# B&R Automation Studio project BaseProject (part 5)

#### Main.st - Init, cyclic, exit code
```iecst
// --------------------------------------------------------------------------------------------------------------------
// Logbook Task
// This task reads the PLC logbook and creates the data structure to display it in mappView
// --------------------------------------------------------------------------------------------------------------------
PROGRAM _INIT
	// Set time range to all on startup
	DTGetTime_0.enable := TRUE;
	DTGetTime_0();
	LogbookInterface.Par.FilterDateStart := STRING_TO_DATE('D#1999-12-31');
	LogbookInterface.Par.FilterDateEnd := DT_TO_DATE(DTGetTime_0.DT1);

	// Read data after reboot
	LogbookInterface.Cmd.Refresh := TRUE;

	// define what object type should be searched for
	LogbookInterface.SegError.ParaSegFilter		:= 'Asm';//'gSeg_';
END_PROGRAM

PROGRAM _CYCLIC
	// Abort current update run
	IF EDGENEG(LogbookInterface.Cmd.Refresh) THEN
		IF 	LogbookState <> STATE_ERROR THEN
			LogbookInterface.Status := ERR_OK;
			LogbookState := STATE_WAIT;
		END_IF
	END_IF

	IF EDGEPOS(DiagInterface.TrakInterface.Asm.Status.ErrorStop) THEN
		LogbookInterface.Cmd.Update := TRUE;
	END_IF

	// Run task multiple times to speed up process
	FOR executions:=1 TO LOGBOOK_EXECUTIONS DO
		// --------------------------------------------------------------------------------------------------------------------
		// Logbook State machine
		// --------------------------------------------------------------------------------------------------------------------
		CASE LogbookState OF
			// --------------------------------------------------------------------------------------------------------------------
			// Wait for new command
			// --------------------------------------------------------------------------------------------------------------------
			STATE_WAIT:
				// --------------------------------------------------------------------------------------------------------------------
				// Get current date
				DTGetTime_0.enable := TRUE;
				DTGetTime_0();
				LogbookInterface.Par.DateNow := DTGetTime_0.DT1;
				LogbookInterface.Par.EntriesMax := LOGBOOK_ENTRIES_MAX;

				// --------------------------------------------------------------------------------------------------------------------
				// Refresh all logbook data
				IF LogbookInterface.Cmd.Refresh THEN
					// Erase old data, set busy state
					brsmemset(ADR(Logbook), 0, SIZEOF(Logbook));
					brsmemset(ADR(LogbookInterface.Data), 0, SIZEOF(LogbookInterface.Data));
					LogbookInterface.Status := ERR_FUB_BUSY;
					LogbookState := STATE_OPEN;
				END_IF

				// --------------------------------------------------------------------------------------------------------------------
				// Auto update logbook data
				IF LogbookInterface.Par.AutoUpdate THEN
					AutoRefresh.IN := TRUE;
					AutoRefresh.PT := LogbookInterface.Par.AutoUpdateInterval*100;
					AutoRefresh();
					IF AutoRefresh.Q THEN
						AutoRefresh(IN:= FALSE);
						LogbookInterface.Cmd.Update := TRUE;
						LogbookState := STATE_NEXT;
					END_IF
				ELSE
					AutoRefresh(IN:= FALSE);
				END_IF

				// --------------------------------------------------------------------------------------------------------------------
				// Update only latest logbook data
				IF LogbookInterface.Cmd.Update THEN
					brsmemset(ADR(Logbook.RecordIDIsLast), 0, SIZEOF(Logbook.RecordIDIsLast));
					brsmemset(ADR(Logbook.RecordID), 0, SIZEOF(Logbook.RecordID));

					brsmemset(ADR(LogbookInterface.SegError.Record), 0, SIZEOF(LogbookInterface.SegError.Record));
					LogbookInterface.SegError.Message := '';
					SegmentErrorFound := 0;

					brsmemset(ADR(AlarmCount), 0, SIZEOF(AlarmCount));

					// Start at the beginning set busy state
					Logbook.CntLogbook := 0;
					LogbookInterface.Status := ERR_FUB_BUSY;
					LogbookState := STATE_LATEST;
				END_IF

				// --------------------------------------------------------------------------------------------------------------------
				// Create new logbook entry
				IF LogbookInterface.Cmd.Create THEN
					LogbookInterface.Status := ERR_FUB_BUSY;
					LogbookState := STATE_CREATE;
				END_IF

				// --------------------------------------------------------------------------------------------------------------------
				// Reset function blocks
				ArEventLogGetIdent_0(Execute := FALSE);
				ArEventLogGetLatestRecordID_0(Execute := FALSE);
				ArEventLogGetPreviousRecordID_0(Execute := FALSE);
				ArEventLogRead_0(Execute := FALSE);
				ArEventLogReadErrorNumber_0(Execute := FALSE);
				ArEventLogReadDescription_0(Execute := FALSE);
				ArEventLogReadAddData_0(Execute := FALSE);
				ArEventLogWrite_0(Execute := FALSE);
				ArEventLogReadObjectID_0(Execute := FALSE);

				// --------------------------------------------------------------------------------------------------------------------
				// Show status, reset error command
				LogbookInterface.Cmd.ResetError := FALSE;
				LogbookInterface.StatusText := 'Waiting...last update ';
				brsstrcat(ADR(LogbookInterface.StatusText), ADR(LogbookInterface.Data.LastUpdate));
				EXIT;
				// --------------------------------------------------------------------------------------------------------------------
				// Create a new logbook entry
				// --------------------------------------------------------------------------------------------------------------------
			STATE_CREATE:
				eventID := ArEventLogMakeEventID(UDINT_TO_USINT(LogbookInterface.Par.CreateSeverity), 0 , LogbookInterface.Par.CreateErrorNo);
				brsmemset(ADR(AddData), 0, SIZEOF(AddData));
				brsstrcpy(ADR(AddData), ADR(LogbookInterface.Par.CreateErrorText));

				ArEventLogWrite_0.Execute := TRUE;
				ArEventLogWrite_0.Ident := Logbook.Ident[LogbookInterface.Par.CreateLogbook];
				ArEventLogWrite_0.EventID := eventID;
				ArEventLogWrite_0.ObjectID := 'User event';
				ArEventLogWrite_0.AddDataFormat := arEVENTLOG_ADDFORMAT_TEXT;
				ArEventLogWrite_0.AddData := ADR(AddData);
				ArEventLogWrite_0.AddDataSize := brsstrlen(ADR(AddData));
				ArEventLogWrite_0();

				// Success
				IF ArEventLogWrite_0.Done AND ArEventLogWrite_0.StatusID = ERR_OK THEN
					ArEventLogWrite_0(Execute := FALSE);
					LogbookInterface.Cmd.Create := FALSE;
					LogbookInterface.Cmd.Update := TRUE;
					LogbookState := STATE_WAIT;
				// Error
				ELSIF ArEventLogWrite_0.Error THEN
					LogbookInterface.Error.State := LogbookState;
					LogbookInterface.Status := ArEventLogWrite_0.StatusID;
					LogbookState := STATE_ERROR;
				END_IF
				// --------------------------------------------------------------------------------------------------------------------
				// Open logbook
				// --------------------------------------------------------------------------------------------------------------------
			STATE_OPEN:
				// Last logbook reached
				IF Logbook.CntLogbook > LOGBOOK_BOOKS_MAX THEN
					Logbook.CntLogbook := 0;
					LogbookState := STATE_LATEST;
					EXIT;
				END_IF
				ArEventLogGetIdent_0.Execute := LogbookInterface.Cmd.Refresh;
				ArEventLogGetIdent_0.Name := LOGBOOK_NAMES[Logbook.CntLogbook];
				ArEventLogGetIdent_0();

				// Success
				IF (ArEventLogGetIdent_0.Done AND ArEventLogGetIdent_0.StatusID = ERR_OK) OR ArEventLogGetIdent_0.StatusID = arEVENTLOG_ERR_LOGBOOK_NOT_FOUND THEN
					Logbook.Ident[Logbook.CntLogbook] := ArEventLogGetIdent_0.Ident;
					Logbook.CntLogbook := Logbook.CntLogbook + 1;
					ArEventLogGetIdent_0(Execute := FALSE);
					// Error
				ELSIF ArEventLogGetIdent_0.Error THEN
					LogbookInterface.Error.State := LogbookState;
					LogbookInterface.Status := ArEventLogGetIdent_0.StatusID;
					LogbookState := STATE_ERROR;
				END_IF
				// --------------------------------------------------------------------------------------------------------------------
				// Read latest entry
				// --------------------------------------------------------------------------------------------------------------------
			STATE_LATEST:
				ArEventLogGetLatestRecordID_0.Execute := TRUE;
				ArEventLogGetLatestRecordID_0.Ident := Logbook.Ident[Logbook.CntLogbook];
				ArEventLogGetLatestRecordID_0();

				// Success
				IF ArEventLogGetLatestRecordID_0.Done AND ArEventLogGetLatestRecordID_0.StatusID = ERR_OK THEN
					// Store this record ID for next step
					Logbook.RecordID[Logbook.CntLogbook] := ArEventLogGetLatestRecordID_0.RecordID;
					// If there is a new entry
					IF ArEventLogGetLatestRecordID_0.RecordID > Logbook.RecordIDOld[Logbook.CntLogbook] THEN
						// Store latest ID for next update command, reset is last flag
						Logbook.RecordIDLatest[Logbook.CntLogbook] := ArEventLogGetLatestRecordID_0.RecordID;
						LogbookState := STATE_DETAILS_1;
						// No new entry
					ELSE
						Logbook.RecordIDIsLast[Logbook.CntLogbook] := TRUE;
						LogbookState := STATE_PREP;
					END_IF
					// Error
				ELSIF ArEventLogGetLatestRecordID_0.Error THEN
					LogbookInterface.Error.State := LogbookState;
					LogbookInterface.Status := ArEventLogGetLatestRecordID_0.StatusID;
					LogbookState := STATE_ERROR;
				END_IF
				// --------------------------------------------------------------------------------------------------------------------
				// Read next entry
				// --------------------------------------------------------------------------------------------------------------------
			STATE_NEXT:
				animation := WorkingStatus(ADR(LogbookInterface.StatusText), ADR('reading entries...'), animation);
				ArEventLogGetPreviousRecordID_0.Execute := TRUE;
				ArEventLogGetPreviousRecordID_0.Ident := Logbook.Ident[Logbook.CntLogbook];
				ArEventLogGetPreviousRecordID_0.RecordID := Logbook.RecordID[Logbook.CntLogbook];
				ArEventLogGetPreviousRecordID_0();

				// Success
				IF ArEventLogGetPreviousRecordID_0.Done AND ArEventLogGetPreviousRecordID_0.StatusID = ERR_OK THEN
					// Store this record ID for next step
					Logbook.RecordID[Logbook.CntLogbook] := ArEventLogGetPreviousRecordID_0.PrevRecordID;
					// Stop update when previous record ID is reached
					IF Logbook.RecordID[Logbook.CntLogbook] = Logbook.RecordIDOld[Logbook.CntLogbook] AND LogbookInterface.Cmd.Update THEN
						// Remember latest entry, set is last flag
						Logbook.RecordIDOld[Logbook.CntLogbook] := Logbook.RecordIDLatest[Logbook.CntLogbook];
						Logbook.RecordIDIsLast[Logbook.CntLogbook] := TRUE;
						LogbookState := STATE_PREP;
					ELSE
						LogbookState := STATE_DETAILS_1;
					END_IF
					// Error
				ELSIF ArEventLogGetPreviousRecordID_0.Error THEN
					// Last entry reached is not an error
					IF ArEventLogGetPreviousRecordID_0.StatusID = arEVENTLOG_ERR_RECORDID_INVALID THEN
						// Remember latest entry, set is last flag
						Logbook.RecordIDOld[Logbook.CntLogbook] := Logbook.RecordIDLatest[Logbook.CntLogbook];
						Logbook.RecordIDIsLast[Logbook.CntLogbook] := TRUE;
						LogbookState := STATE_PREP;
						// Everything else is an error
					ELSE
						LogbookInterface.Error.State := LogbookState;
						LogbookInterface.Status := ArEventLogGetPreviousRecordID_0.StatusID;
						LogbookState := STATE_ERROR;
					END_IF
				END_IF
				// --------------------------------------------------------------------------------------------------------------------
				// Read event id and time stamp
				// --------------------------------------------------------------------------------------------------------------------
			STATE_DETAILS_1:
				ArEventLogRead_0.Execute := TRUE;
				ArEventLogRead_0.Ident := Logbook.Ident[Logbook.CntLogbook];
				ArEventLogRead_0.RecordID := Logbook.RecordID[Logbook.CntLogbook];
				ArEventLogRead_0();

				// Success
				IF ArEventLogRead_0.Done AND (ArEventLogRead_0.StatusID = ERR_OK OR ArEventLogRead_0.StatusID = arEVENTLOG_WRN_NO_EVENTID) THEN
					LogbookState := STATE_DETAILS_2;

					EventID := ArEventLogRead_0.EventID;
					EventTimeStamp := ArEventLogRead_0.TimeStamp;
					EventIDSeverity	:= DINT_TO_USINT(SHR(EventID, 30) AND 16#03);
					EventIDFacility	:= DINT_TO_UINT(SHR(EventID, 16) AND 16#0FFF);
					EventIDCode		:= DINT_TO_UINT(SHR(EventID, 0) AND 16#FFFF);

				// Error
				ELSIF ArEventLogRead_0.Error THEN
					LogbookInterface.Error.State := LogbookState;
					LogbookInterface.Status := ArEventLogRead_0.StatusID;
					LogbookState := STATE_ERROR;
				END_IF
				// --------------------------------------------------------------------------------------------------------------------
				// Read error no
				// --------------------------------------------------------------------------------------------------------------------
			STATE_DETAILS_2:
				ArEventLogReadErrorNumber_0.Execute := TRUE;
				ArEventLogReadErrorNumber_0.Ident := Logbook.Ident[Logbook.CntLogbook];
				ArEventLogReadErrorNumber_0.RecordID := Logbook.RecordID[Logbook.CntLogbook];
				ArEventLogReadErrorNumber_0();

				// Success
				IF (ArEventLogReadErrorNumber_0.Done AND ArEventLogReadErrorNumber_0.StatusID = ERR_OK) OR ArEventLogReadErrorNumber_0.StatusID = arEVENTLOG_ERR_NO_ERRORNUMBER THEN
					brsmemset(ADR(ErrorText), 0, SIZEOF(ErrorText));
					LogbookState := STATE_DETAILS_3;
				// Error
				ELSIF ArEventLogReadErrorNumber_0.Error THEN
					LogbookInterface.Error.State := LogbookState;
					LogbookInterface.Status := ArEventLogReadErrorNumber_0.StatusID;
					LogbookState := STATE_ERROR;
				END_IF
				// --------------------------------------------------------------------------------------------------------------------
				// Read error description
				// --------------------------------------------------------------------------------------------------------------------
			STATE_DETAILS_3:
				ArEventLogReadDescription_0.Execute := TRUE;
				ArEventLogReadDescription_0.Ident := Logbook.Ident[Logbook.CntLogbook];
				ArEventLogReadDescription_0.RecordID := Logbook.RecordID[Logbook.CntLogbook];
				ArEventLogReadDescription_0.TextBuffer := ADR(ErrorText);
				ArEventLogReadDescription_0.TextBufferSize := SIZEOF(ErrorText);
				ArEventLogReadDescription_0();

				// Success
				IF (ArEventLogReadDescription_0.Done AND (ArEventLogReadDescription_0.StatusID = ERR_OK OR ArEventLogReadDescription_0.StatusID = arEVENTLOG_WRN_NO_EVENTID)) OR ArEventLogReadDescription_0.StatusID = arEVENTLOG_ERR_NO_DESCRIPTION THEN
					brsmemset(ADR(AddData), 0, SIZEOF(AddData));
					IF ((Logbook.CntLogbook = 6) AND (EventIDSeverity = arEVENTLOG_SEVERITY_ERROR)) THEN (*6 = index for motion logbook*)
						LogbookState := STATE_CHECK_FILTER;
					ELSE
						LogbookState := STATE_DETAILS_4;
					END_IF
				// Error
				ELSIF ArEventLogReadDescription_0.Error THEN
					LogbookInterface.Error.State := LogbookState;
					LogbookInterface.Status := ArEventLogReadDescription_0.StatusID;
					LogbookState := STATE_ERROR;
				END_IF

			///////////////////////////////////////////////////////////////////////////
			// check if 'Error' has been entered by a Segment
			STATE_CHECK_FILTER:
				ArEventLogReadObjectID_0.Execute	:= TRUE;
				ArEventLogReadObjectID_0.Ident		:= Logbook.Ident[Logbook.CntLogbook];
				ArEventLogReadObjectID_0.RecordID	:= Logbook.RecordID[Logbook.CntLogbook];
				ArEventLogReadObjectID_0();

				IF ArEventLogReadObjectID_0.Done THEN
					ObjectID := ArEventLogReadObjectID_0.ObjectID;
					ArEventLogReadObjectID_0.Execute := FALSE;
					IF brsmemcmp(ADR(ObjectID), ADR(LogbookInterface.SegError.ParaSegFilter), 3) = 0 THEN
						LogbookState := STATE_UPDATE_LIST;
					ELSE
						LogbookState := STATE_DETAILS_4;
					END_IF
				ELSIF ArEventLogReadObjectID_0.Error THEN
					LogbookInterface.SegError.Message := 'Error ReadObjectID';
					LogbookState := STATE_ERROR;
				END_IF

			STATE_UPDATE_LIST:
				LogbookInterface.SegError.Record[SegmentErrorFound].ObjectID		:= ObjectID;
				LogbookInterface.SegError.Record[SegmentErrorFound].EventID			:= EventID;
				LogbookInterface.SegError.Record[SegmentErrorFound].EventIDSeverity	:= EventIDSeverity;
				LogbookInterface.SegError.Record[SegmentErrorFound].EventIDFacility	:= EventIDFacility;
				LogbookInterface.SegError.Record[SegmentErrorFound].EventIDCode		:= EventIDCode;
				LogbookInterface.SegError.Record[SegmentErrorFound].Description		:= Description;

				LogbookInterface.SegError.Record[SegmentErrorFound].EventTimeStamp	:= UDINT_TO_TIME((EventTimeStamp.sec MOD (24*60*60))*1000 + (EventTimeStamp.nsec / 1000000));		// convert to TIME format (ms since start of day)

				brsstrcpy(ADR(LogbookInterface.SegError.Record[SegmentErrorFound].Text), ADR(''));
				ascTIME(LogbookInterface.SegError.Record[SegmentErrorFound].EventTimeStamp, ADR(TempString), SIZEOF(TempString));
				TIME_TO_TIMEStructure(LogbookInterface.SegError.Record[SegmentErrorFound].EventTimeStamp,ADR(TimeStruct)); // for checking against older entries

				brsstrcat(ADR(LogbookInterface.SegError.Record[SegmentErrorFound].Text), ADR(TempString));
				brsstrcat(ADR(LogbookInterface.SegError.Record[SegmentErrorFound].Text), ADR(' => '));

				brsstrcat(ADR(LogbookInterface.SegError.Record[SegmentErrorFound].Text), ADR(ObjectID));

				brsstrcat(ADR(LogbookInterface.SegError.Record[SegmentErrorFound].Text), ADR(': Error '));
				brsitoa(EventIDCode, ADR(TempString));
				brsstrcat(ADR(LogbookInterface.SegError.Record[SegmentErrorFound].Text), ADR(TempString));

				brsstrcat(ADR(LogbookInterface.SegError.Record[SegmentErrorFound].Text), ADR(' => '));
				brsstrcat(ADR(LogbookInterface.SegError.Record[SegmentErrorFound].Text), ADR(Description));

				IF SegmentErrorFound = 0 THEN
					FirstEntryCheckSum := TimeStruct.minute; // save the timestamp minute of the first entry as checksum
				END_IF

				SegmentErrorFound := SegmentErrorFound + 1;

				SetTrakSegAlarm(DiagInterface.AlarmCore,EventIDCode,ADR(AlarmCount));

				// stop reading the logger when the end of the array is reached OR
				// when the entries start having a different timestamp which means they are older
				IF SegmentErrorFound > 499 OR (FirstEntryCheckSum <> (TimeStruct.minute) ) THEN
					LogbookState := STATE_DETAILS_4;
				ELSE
					LogbookState := STATE_DETAILS_4;
				END_IF

				// --------------------------------------------------------------------------------------------------------------------
				// Read additional information
				// --------------------------------------------------------------------------------------------------------------------
			STATE_DETAILS_4:
				// Skip if no additional data is available
				IF ArEventLogRead_0.AddDataSize > 0 THEN
					// Read additional data
					ArEventLogReadAddData_0.Execute := TRUE;
					ArEventLogReadAddData_0.Ident := Logbook.Ident[Logbook.CntLogbook];
					ArEventLogReadAddData_0.RecordID := Logbook.RecordID[Logbook.CntLogbook];
					ArEventLogReadAddData_0.AddData := ADR(AddData);
					// Limit buffer to max size
					IF ArEventLogRead_0.AddDataSize < SIZEOF(AddData) THEN
						ArEventLogReadAddData_0.BytesToRead := ArEventLogRead_0.AddDataSize;
					ELSE
						ArEventLogReadAddData_0.BytesToRead := SIZEOF(AddData);
					END_IF
					ArEventLogReadAddData_0();

					// Success
					IF (ArEventLogReadAddData_0.Done AND ArEventLogReadAddData_0.StatusID = ERR_OK) OR ArEventLogReadAddData_0.StatusID = arEVENTLOG_INF_SIZE THEN
						// Enter standard text if additional does not fit
						IF ArEventLogReadAddData_0.StatusID = arEVENTLOG_INF_SIZE THEN
							brsstrcat(ADR(ErrorText), ADR('\n >>> '));
							brsstrcat(ADR(ErrorText), ADR('Additional buffer is too small'));
						ELSE
							// Make sure string is readable
							IF brsstrcmp(ADR(AddData), ADR('')) <> 0 AND ArEventLogRead_0.AddDataFormat = arEVENTLOG_ADDFORMAT_TEXT THEN
								brsstrcat(ADR(ErrorText), ADR('\n >>> '));
								// Limit additional text to max size
								IF ArEventLogReadAddData_0.AddDataSize < SIZEOF(ErrorText) - brsstrlen(ADR(ErrorText)) THEN
									brsstrcat(ADR(ErrorText), ADR(AddData));
								ELSE
									brsmemcpy(ADR(ErrorText) + brsstrlen(ADR(ErrorText)), ADR(AddData), SIZEOF(ErrorText) - brsstrlen(ADR(ErrorText)));
								END_IF
							END_IF
						END_IF
						LogbookState := STATE_FILTER;
					// Error
					ELSIF ArEventLogReadDescription_0.Error THEN
						LogbookInterface.Error.State := LogbookState;
						LogbookInterface.Status := ArEventLogReadAddData_0.StatusID;
						LogbookState := STATE_ERROR;
					END_IF
				ELSE
					LogbookState := STATE_FILTER;
				END_IF
				// --------------------------------------------------------------------------------------------------------------------
				// Apply filter settings
				// --------------------------------------------------------------------------------------------------------------------
			STATE_FILTER:
				// --------------------------------------------------------------------------------------------------------------------
				// Filters
				cntFilterNo := 0;
				cntFilterText := 0;
				cntFilterLogbook := 0;
				cntFilterSeverity := 0;
				cntFilterDate := 0;
				// --------------------------------------------------------------------------------------------------------------------
				// Check if logbook should be read
				IF  LogbookInterface.Par.FilterLogbook[Logbook.CntLogbook] THEN
					cntFilterLogbook := cntFilterLogbook + 1;
				END_IF
				// --------------------------------------------------------------------------------------------------------------------
				// Check if error text matches search string
				IF LogbookInterface.Par.FilterErrorText = '' OR IsInstr(ADR(ErrorText), ADR(LogbookInterface.Par.FilterErrorText)) THEN
					cntFilterText := cntFilterText + 1;
				END_IF
				// --------------------------------------------------------------------------------------------------------------------
				// Make sure error number matches filter
				IF LogbookInterface.Par.FilterErrorNo = 0 OR LogbookInterface.Par.FilterErrorNo = ArEventLogReadErrorNumber_0.ErrorNumber THEN
					cntFilterNo := cntFilterNo + 1;
				END_IF
				// --------------------------------------------------------------------------------------------------------------------
				// Check severity filter settings
				IF ArEventLogRead_0.EventID <> 0 THEN
					LogbookInterface.Data.CntSeverity[GetSeverity(EventID := ArEventLogRead_0.EventID)] := LogbookInterface.Data.CntSeverity[GetSeverity(EventID := ArEventLogRead_0.EventID)] + 1;
					IF LogbookInterface.Par.FilterSeverity[GetSeverity(EventID := ArEventLogRead_0.EventID)] THEN
						cntFilterSeverity := cntFilterSeverity + 1;
					END_IF
				ELSE
					LogbookInterface.Data.CntSeverity[ArEventLogReadErrorNumber_0.Severity] := LogbookInterface.Data.CntSeverity[ArEventLogReadErrorNumber_0.Severity] + 1;
					IF LogbookInterface.Par.FilterSeverity[ArEventLogReadErrorNumber_0.Severity] THEN
						cntFilterSeverity := cntFilterSeverity + 1;
					END_IF
				END_IF
				// --------------------------------------------------------------------------------------------------------------------
				// Check date range
				tmpSTR:= DT_TO_STRING(DATE_TO_DT(LogbookInterface.Par.FilterDateStart));
				brsmemcpy(ADR(tmpSTR)+13, ADR('-00:00:00'), 9);
				TimeStart := STRING_TO_DT(tmpSTR);
				tmpSTR:= DT_TO_STRING(DATE_TO_DT(LogbookInterface.Par.FilterDateEnd));
				brsmemcpy(ADR(tmpSTR)+13, ADR('-23:59:59'), 9);
				TimeEnd := STRING_TO_DT(tmpSTR);
				IF ArEventLogRead_0.TimeStamp.sec >= DT_TO_UDINT(TimeStart) AND ArEventLogRead_0.TimeStamp.sec <= DT_TO_UDINT(TimeEnd) THEN
					cntFilterDate := cntFilterDate + 1;
				END_IF
				// --------------------------------------------------------------------------------------------------------------------
				// Count logbook entries
				LogbookInterface.Data.CntLogbook[Logbook.CntLogbook] := LogbookInterface.Data.CntLogbook[Logbook.CntLogbook] +  1;

				// --------------------------------------------------------------------------------------------------------------------
				// Transfer data
				IF cntFilterNo > 0 AND cntFilterText > 0 AND cntFilterLogbook > 0 AND cntFilterSeverity > 0 AND cntFilterDate > 0 THEN
					// --------------------------------------------------------------------------------------------------------------------
					// Find new place for entry
					idx := InsertEntry(ADR(LogbookInterface.Data), ArEventLogRead_0.TimeStamp.sec, UDINT_TO_UINT(ArEventLogRead_0.TimeStamp.nsec/1000000), LogbookInterface.Par.Sorting);
					IF idx <> NO_SPACE THEN
						// Store date and time
						LogbookInterface.Data.Entries.DTsec[idx] := ArEventLogRead_0.TimeStamp.sec;
						LogbookInterface.Data.Entries.DTmsec[idx] := UDINT_TO_UINT(ArEventLogRead_0.TimeStamp.nsec/1000000);
						// Add timestamp
						tmpDT := UDINT_TO_DT(ArEventLogRead_0.TimeStamp.sec);
						DT_TO_DTStructure(tmpDT, ADR(tmpDTstruct));
						brsmemset(ADR(LogbookInterface.Data.Entries.Timestamp[idx]), 0, SIZEOF(LogbookInterface.Data.Entries.Timestamp[idx]));
						NormalizeDateTime(ADR(LogbookInterface.Data.Entries.Timestamp[idx]), tmpDTstruct.day, '');
						NormalizeDateTime(ADR(LogbookInterface.Data.Entries.Timestamp[idx]), tmpDTstruct.month, '.');
						NormalizeDateTime(ADR(LogbookInterface.Data.Entries.Timestamp[idx]), tmpDTstruct.year, '.');
						NormalizeDateTime(ADR(LogbookInterface.Data.Entries.Timestamp[idx]), tmpDTstruct.hour, ' ');
						NormalizeDateTime(ADR(LogbookInterface.Data.Entries.Timestamp[idx]), tmpDTstruct.minute, ':');
						NormalizeDateTime(ADR(LogbookInterface.Data.Entries.Timestamp[idx]), tmpDTstruct.second, ':');
						NormalizeDateTime(ADR(LogbookInterface.Data.Entries.Timestamp[idx]), LogbookInterface.Data.Entries.DTmsec[idx], '.');
						// Add event ID, code, logbook, severity
						LogbookInterface.Data.Entries.EventID[LogbookInterface.Data.EntriesTotal] := ArEventLogRead_0.EventID;
						IF ArEventLogRead_0.EventID <> 0 THEN
							LogbookInterface.Data.Entries.Severity[idx] := GetSeverity(EventID := ArEventLogRead_0.EventID);
						ELSE
							LogbookInterface.Data.Entries.Severity[idx] := ArEventLogReadErrorNumber_0.Severity;
						END_IF
						LogbookInterface.Data.Entries.Code[idx] := GetCode(EventID := ArEventLogRead_0.EventID);
						LogbookInterface.Data.Entries.FacilityCode[idx] := GetFacility(EventID := ArEventLogRead_0.EventID);
						LogbookInterface.Data.Entries.LogbookName[idx] := LOGBOOK_TEXT[Logbook.CntLogbook];
						// Add error number and text, use event ID if error no is 0
						IF ArEventLogReadErrorNumber_0.ErrorNumber <> 0 THEN
							LogbookInterface.Data.Entries.ErrorNo[idx] := ArEventLogReadErrorNumber_0.ErrorNumber;
						ELSE
							LogbookInterface.Data.Entries.ErrorNo[idx] := ArEventLogRead_0.EventID;
						END_IF
						httpUtf8ToString_0(enable := TRUE, pSrc := ADR(ErrorText), pDest := ADR(LogbookInterface.Data.Entries.ErrorText[idx]), destSize := SIZEOF(LogbookInterface.Data.Entries.ErrorText[idx]));
					END_IF
				END_IF

				// --------------------------------------------------------------------------------------------------------------------
				// Hide unused table rows
				brsitoa(LogbookInterface.Data.EntriesTotal, ADR(tmpSTR));
				LogbookInterface.Par.TableConfig := '{"specRows":[{"from":';
				brsstrcat(ADR(LogbookInterface.Par.TableConfig), ADR(tmpSTR));
				brsstrcat(ADR(LogbookInterface.Par.TableConfig), ADR(', "to":'));
				brsitoa(LOGBOOK_ENTRIES_MAX, ADR(tmpSTR));
				brsstrcat(ADR(LogbookInterface.Par.TableConfig), ADR(tmpSTR));
				brsstrcat(ADR(LogbookInterface.Par.TableConfig), ADR(', "visible":false}]}'));

				LogbookState := STATE_PREP;

				// --------------------------------------------------------------------------------------------------------------------
				// Perpare for next entry
				// --------------------------------------------------------------------------------------------------------------------
			STATE_PREP:
				// --------------------------------------------------------------------------------------------------------------------
				// Reset buffer and function blocks
				brsmemset(ADR(AddData), 0, SIZEOF(AddData));
				ArEventLogGetLatestRecordID_0(Execute := FALSE);
				ArEventLogGetPreviousRecordID_0(Execute := FALSE);
				ArEventLogRead_0(Execute := FALSE);
				ArEventLogReadErrorNumber_0(Execute := FALSE);
				ArEventLogReadDescription_0(Execute := FALSE);
				ArEventLogReadAddData_0(Execute := FALSE);
				ArEventLogReadObjectID_0(Execute := FALSE);

				// --------------------------------------------------------------------------------------------------------------------
				// Find next logbook from here to the end
				REPEAT
					Logbook.CntLogbook := Logbook.CntLogbook + 1;
					IF Logbook.CntLogbook <= LOGBOOK_BOOKS_MAX THEN
						IF (Logbook.Ident[Logbook.CntLogbook] <> 0 AND NOT Logbook.RecordIDIsLast[Logbook.CntLogbook]) OR (Logbook.Ident[Logbook.CntLogbook] <> 0 AND Logbook.RecordID[Logbook.CntLogbook] = 0) THEN
							EXIT;
						END_IF
					END_IF
					UNTIL Logbook.CntLogbook > LOGBOOK_BOOKS_MAX
				END_REPEAT;

				// --------------------------------------------------------------------------------------------------------------------
				// No logbook found, start at the beginning
				IF Logbook.CntLogbook > LOGBOOK_BOOKS_MAX THEN
					Logbook.CntLogbook := 0;
					// Find next logbook from start to the end
					REPEAT
						IF (Logbook.Ident[Logbook.CntLogbook] <> 0 AND NOT Logbook.RecordIDIsLast[Logbook.CntLogbook]) OR (Logbook.Ident[Logbook.CntLogbook] <> 0 AND Logbook.RecordID[Logbook.CntLogbook] = 0) THEN
							EXIT;
						END_IF
						Logbook.CntLogbook := Logbook.CntLogbook + 1;
						UNTIL Logbook.CntLogbook > LOGBOOK_BOOKS_MAX
					END_REPEAT;
				END_IF

				// --------------------------------------------------------------------------------------------------------------------
				// Finish when no logbook found or max entries is reached
				IF Logbook.CntLogbook > LOGBOOK_BOOKS_MAX OR (LogbookInterface.Par.AbortOnEntriesLimit AND LogbookInterface.Data.EntriesTotal = LOGBOOK_ENTRIES_MAX) THEN
					// Add last update
					DT_TO_DTStructure(LogbookInterface.Par.DateNow, ADR(tmpDTstruct));
					brsmemset(ADR(LogbookInterface.Data.LastUpdate), 0, SIZEOF(LogbookInterface.Data.LastUpdate));
					NormalizeDateTime(ADR(LogbookInterface.Data.LastUpdate), tmpDTstruct.day, '');
					NormalizeDateTime(ADR(LogbookInterface.Data.LastUpdate), tmpDTstruct.month, '.');
					NormalizeDateTime(ADR(LogbookInterface.Data.LastUpdate), tmpDTstruct.year, '.');
					NormalizeDateTime(ADR(LogbookInterface.Data.LastUpdate), tmpDTstruct.hour, ' ');
					NormalizeDateTime(ADR(LogbookInterface.Data.LastUpdate), tmpDTstruct.minute, ':');
					NormalizeDateTime(ADR(LogbookInterface.Data.LastUpdate), tmpDTstruct.second, ':');
					// Reset status and command
					LogbookInterface.Status := ERR_OK;
					LogbookInterface.Cmd.Refresh := FALSE;
					LogbookInterface.Cmd.Update := FALSE;
					LogbookState := STATE_WAIT;
				ELSE
					// Read latest entry
					IF Logbook.RecordID[Logbook.CntLogbook] = 0 THEN
						LogbookState := STATE_LATEST;
						// Read next entry
					ELSE
						LogbookState := STATE_NEXT;
					END_IF
				END_IF

				// --------------------------------------------------------------------------------------------------------------------
				// Error state
				// --------------------------------------------------------------------------------------------------------------------
			STATE_ERROR:
				LogbookInterface.StatusText := 'Error...';
				brsmemset(ADR(LogbookInterface.Cmd), 0, SIZEOF(LogbookInterface.Cmd)-1);
				// Reset error
				IF LogbookInterface.Cmd.ResetError THEN
					LogbookInterface.Error.State := STATE_NONE;
					LogbookInterface.Status := 0;
					LogbookInterface.Cmd.ResetError := FALSE;
					LogbookState := STATE_WAIT;
				END_IF
				EXIT;
		END_CASE;
	END_FOR;

END_PROGRAM
```

#### Variables.var - Local variables
```iecst
(*---------------------------------------------------------------------------------------------------------------------------------*)
VAR
	ErrorText : STRING[LOGBOOK_TEXT_LEN];
	cntFilterNo : UINT;
	cntFilterText : UINT;
	cntFilterLogbook : UINT;
	cntFilterSeverity : UINT;
	cntFilterDate : UINT;
	tmpSTR : STRING[100];
	tmpDT : DATE_AND_TIME;
	tmpDTstruct : DTStructure;
	TimeStart : DATE_AND_TIME;
	TimeEnd : DATE_AND_TIME;
	AddData : ARRAY[0..500] OF USINT;
	Logbook : LogBooksType;
	idx : UINT;
	eventID : DINT;
	animation : USINT;
END_VAR
(*---------------------------------------------------------------------------------------------------------------------------------*)
(*Local function*)
VAR
	ArEventLogGetPreviousRecordID_0 : ArEventLogGetPreviousRecordID;
	ArEventLogGetLatestRecordID_0 : ArEventLogGetLatestRecordID;
	ArEventLogRead_0 : ArEventLogRead;
	ArEventLogWrite_0 : ArEventLogWrite;
	ArEventLogReadErrorNumber_0 : ArEventLogReadErrorNumber;
	ArEventLogReadDescription_0 : ArEventLogReadDescription;
	ArEventLogReadAddData_0 : ArEventLogReadAddData;
	ArEventLogReadObjectID_0 : ArEventLogReadObjectID;
	DTGetTime_0 : DTGetTime;
	httpUtf8ToString_0 : httpUtf8ToString;
	AutoRefresh : TON_10ms;
END_VAR
(*Local variables*)
VAR
	LogbookState : LogBookStateEnum;
	ArEventLogGetIdent_0 : ArEventLogGetIdent;
	executions : USINT;
END_VAR
(*---------------------------------------------------------------------------------------------------------------------------------*)
(*Local constants*)
VAR CONSTANT
	LOGBOOK_NAMES : ARRAY[0..LOGBOOK_BOOKS_MAX] OF STRING[50] := ['$$accsec','$$diag','$$arlogconn','$$fieldbus','$$firewall','$$mapp','$$motion','$$safety','$$arlogsys','$$textsys','$$unitsys','$$arlogusr','$$vision','$$visu'];
	LOGBOOK_TEXT : ARRAY[0..LOGBOOK_BOOKS_MAX] OF STRING[50] := ['Access','Commissioning','Connectivity','Fieldbus','Firewall','Mapp','Motion','Safety','System','Text System','Unit System','User','Vision','Visualization'];
	NO_SPACE : UINT := 0;
END_VAR
(*read & filter motion logger*)
VAR
	EventID : DINT := 0;
	EventIDSeverity : USINT := 0;
	EventIDFacility : UINT := 0;
	EventIDCode : UINT := 0;
	EventTimeStamp : ArEventLogTimeStampType := (0);
	ObjectID : STRING[36] := '';
	Description : STRING[256] := '';
	TempString : STRING[32] := '';
	SegmentErrorFound : USINT := 0;
	AlarmCount : ARRAY[0..119] OF UDINT;
	TimeStruct : TIMEStructure;
	FirstEntryCheckSum : USINT;
END_VAR
(*Test function*)
VAR
	MC_BR_SegCommandError_AcpTrak_0 : MC_BR_SegCommandError_AcpTrak;
END_VAR
```

#### Types.typ
```iecst
TYPE
	typLogbook : 	STRUCT
		Ident : ARRAY[0..LOGBOOK_BOOKS_MAX]OF UDINT;
		RecordIDLatest : ARRAY[0..LOGBOOK_BOOKS_MAX]OF UDINT;
		RecordIDOld : ARRAY[0..LOGBOOK_BOOKS_MAX]OF UDINT;
		RecordIDIsLast : ARRAY[0..LOGBOOK_BOOKS_MAX]OF BOOL;
		RecordID : ARRAY[0..LOGBOOK_BOOKS_MAX]OF UDINT;
		CntLogbook : USINT;
	END_STRUCT;
END_TYPE
```

#### LocalFunctions.fun
```iecst
FUNCTION GetSeverity : USINT
	VAR_INPUT
		EventID : DINT;
	END_VAR
END_FUNCTION

FUNCTION GetFacility : UINT
	VAR_INPUT
		EventID : DINT;
	END_VAR
END_FUNCTION

{REDUND_ERROR} FUNCTION GetCode : UINT (*create mappView string data provider*) (*$GROUP=User,$CAT=User,$GROUPICON=User.png,$CATICON=User.png*)
	VAR_INPUT
		EventID : DINT;
	END_VAR
END_FUNCTION

FUNCTION InsertEntry : UINT
	VAR_INPUT
		Data : REFERENCE TO LogBookDataType;
		DTsec : UDINT;
		DTmsec : UINT;
		Sorting : LogBookSortingEnum;
	END_VAR
	VAR
		idx : UINT;
		idy : UINT;
	END_VAR
END_FUNCTION

FUNCTION NormalizeDateTime : UDINT
	VAR_INPUT
		Target : UDINT;
		Value : UDINT;
		AddSTR : STRING[5];
	END_VAR
	VAR
		tmpSTR1 : STRING[10];
		tmpSTR2 : STRING[10];
	END_VAR
END_FUNCTION

FUNCTION WorkingStatus : USINT
	VAR_INPUT
		Target : UDINT;
		Text : UDINT;
		Animation : USINT;
	END_VAR
END_FUNCTION

FUNCTION IsInstr : BOOL
	VAR_INPUT
		String1 : UDINT;
		String2 : UDINT;
	END_VAR
	VAR
		idx : UDINT;
	END_VAR
END_FUNCTION

{REDUND_ERROR} FUNCTION SetTrakSegAlarm : BOOL (*Trigger MpAlarmXSet based on EventIDCode*) (*$GROUP=User,$CAT=User,$GROUPICON=User.png,$CATICON=User.png*)
	VAR_INPUT
		AlarmMpLink : MpComIdentType;
		EventIDCode : UDINT;
		AlarmCount : REFERENCE TO ARRAY[0..119] OF UDINT;
	END_VAR
END_FUNCTION
```

#### LocalFunctions.st
```iecst
// --------------------------------------------------------------------------------------------------------------------
// Gets severity from EventId (bits 31-30)
FUNCTION GetSeverity
	IF ArEventLogIsError(EventID := EventID) THEN
		GetSeverity := arEVENTLOG_SEVERITY_ERROR;
	ELSIF ArEventLogIsWarning(EventID := EventID) THEN
		GetSeverity := arEVENTLOG_SEVERITY_WARNING;
	ELSIF ArEventLogIsInformation(EventID := EventID) THEN
		GetSeverity := arEVENTLOG_SEVERITY_INFO;
	ELSIF ArEventLogIsSuccess(EventID := EventID) THEN
		GetSeverity := arEVENTLOG_SEVERITY_SUCCESS;
	END_IF
END_FUNCTION

// --------------------------------------------------------------------------------------------------------------------
// Gets code from EventId (bits 15-0)
FUNCTION GetCode
	GetCode := DINT_TO_UINT(EventID);
END_FUNCTION

// --------------------------------------------------------------------------------------------------------------------
// Gets facility from EventId (bits 27-16)
FUNCTION GetFacility
	GetFacility := DINT_TO_UINT(SHR(EventID, 16) AND 16#0FFF);
END_FUNCTION

// --------------------------------------------------------------------------------------------------------------------
// --------------------------------------------------------------------------------------------------------------------
// Insert new entry
FUNCTION InsertEntry
	// Lets see where new entry fits
	FOR idx:=1 TO DAT.EntriesTotal DO
		// Sorting is ascending
		IF Sorting = SORTING_ASC THEN
			// New entry is old than this entry
			IF DTsec < DAT.Entries.DTsec[idx] THEN
				EXIT;
				// If entries are within the same second check milisecond data
			ELSIF DTsec = DAT.Entries.DTsec[idx] THEN
				IF DTmsec < DAT.Entries.DTmsec[idx] THEN
					EXIT;
				END_IF
			END_IF
			// Sorting is descending
		ELSE
			// New entry is newer than this entry
			IF DTsec > DAT.Entries.DTsec[idx] THEN
				EXIT;
				// If entries are within the same second check milisecond data
			ELSIF DTsec = DAT.Entries.DTsec[idx] THEN
				IF DTmsec > DAT.Entries.DTmsec[idx] THEN
					EXIT;
				END_IF
			END_IF
		END_IF
	END_FOR;

	// Add data as long as buffer is not full
	IF DAT.EntriesTotal < LOGBOOK_ENTRIES_MAX THEN
		IF DAT.EntriesTotal = 1 AND idx = 1 THEN
			idy := 1;
		ELSIF DAT.EntriesTotal >= idx THEN
			idy := DAT.EntriesTotal - idx + 1;
		END_IF
		DAT.EntriesTotal := DAT.EntriesTotal + 1;
		// If buffer is full check where entry fits
	ELSE
		// Entry is beyond scope of buffer
		IF idx > LOGBOOK_ENTRIES_MAX THEN
			InsertEntry := NO_SPACE;
			RETURN;
		ELSE
			IF DAT.EntriesTotal - idx > 0 THEN
				idy := DAT.EntriesTotal - idx;
			END_IF
		END_IF
	END_IF

	// Dont move if there is nothing to move
	IF idy <> 0 THEN
		brsmemmove(ADR(DAT.Entries.Code[idx+1]),ADR(DAT.Entries.Code[idx]), idy * SIZEOF(DAT.Entries.Code[1]));
		brsmemmove(ADR(DAT.Entries.Timestamp[idx+1]),ADR(DAT.Entries.Timestamp[idx]), idy * SIZEOF(DAT.Entries.Timestamp[1]));
		brsmemmove(ADR(DAT.Entries.DTsec[idx+1]),ADR(DAT.Entries.DTsec[idx]), idy * SIZEOF(DAT.Entries.DTsec[1]));
		brsmemmove(ADR(DAT.Entries.DTmsec[idx+1]),ADR(DAT.Entries.DTmsec[idx]), idy * SIZEOF(DAT.Entries.DTmsec[1]));
		brsmemmove(ADR(DAT.Entries.ErrorNo[idx+1]),ADR(DAT.Entries.ErrorNo[idx]), idy * SIZEOF(DAT.Entries.ErrorNo[1]));
		brsmemmove(ADR(DAT.Entries.ErrorText[idx+1]),ADR(DAT.Entries.ErrorText[idx]), idy * SIZEOF(DAT.Entries.ErrorText[1]));
		brsmemmove(ADR(DAT.Entries.EventID[idx+1]),ADR(DAT.Entries.EventID[idx]), idy * SIZEOF(DAT.Entries.EventID[1]));
		brsmemmove(ADR(DAT.Entries.FacilityCode[idx+1]),ADR(DAT.Entries.FacilityCode[idx]), idy * SIZEOF(DAT.Entries.FacilityCode[1]));
		brsmemmove(ADR(DAT.Entries.LogbookName[idx+1]),ADR(DAT.Entries.LogbookName[idx]), idy * SIZEOF(DAT.Entries.LogbookName[1]));
		brsmemmove(ADR(DAT.Entries.Severity[idx+1]),ADR(DAT.Entries.Severity[idx]), idy * SIZEOF(DAT.Entries.Severity[1]));
	END_IF
	InsertEntry := idx;

END_FUNCTION

// --------------------------------------------------------------------------------------------------------------------
// Normalize 2 digit date and time values
FUNCTION NormalizeDateTime
	tmpSTR2 := addSTR;
	IF(value < 10) THEN
		brsstrcat(ADR(tmpSTR2), ADR('0'));
	END_IF
	brsitoa(value, ADR(tmpSTR1));
	brsstrcat(ADR(tmpSTR2), ADR(tmpSTR1));
	brsstrcat(target, ADR(tmpSTR2));
	NormalizeDateTime := TRUE;
END_FUNCTION

// --------------------------------------------------------------------------------------------------------------------
// Working status
FUNCTION WorkingStatus
	animation := animation+1;

	IF (animation = 80) THEN
		animation := 0;
	END_IF

	brsstrcpy(target, text);
	CASE(animation) OF
		0..19	: brsstrcat(target, ADR('/'));
		20..39	: brsstrcat(target, ADR('-'));
		40..59	: brsstrcat(target, ADR('\'));
		60..79	: brsstrcat(target, ADR('|'));
	END_CASE;
	WorkingStatus := animation;
END_FUNCTION

// --------------------------------------------------------------------------------------------------------------------
// Is second string in first string
FUNCTION IsInstr
	IF (brsstrlen(string1) > brsstrlen(string2)) THEN
		FOR idx:=0 TO brsstrlen(string1) - brsstrlen(string2) DO
			IF (brsmemcmp(string1 + idx, string2, brsstrlen(string2)) = 0) THEN
				IsInstr := TRUE;
				EXIT;
			END_IF
		END_FOR;
	END_IF
END_FUNCTION

(* Trigger proper alarms *)
FUNCTION SetTrakSegAlarm

		SetTrakSegAlarm := TRUE;
		// EventIDCode add new alarms triggers at the end otherwise
		// the AlarmCount has to be adjusted not just here but also for all the alarms in the MpAlarmX config

		CASE EventIDCode OF
		// every time the alarm is triggered it's counted so a total count can be displayed in the alarm message
		1	 :  AlarmCount[0  ] :=  AlarmCount[0]  + 1;   MpAlarmXSet(AlarmMpLink,'EventIDCode.1	');
		2	 :  AlarmCount[1  ] :=  AlarmCount[1]  + 1;   MpAlarmXSet(AlarmMpLink,'EventIDCode.2	');
		7	 :  AlarmCount[2  ] :=  AlarmCount[2]  + 1;   MpAlarmXSet(AlarmMpLink,'EventIDCode.7	');
		2048 :  AlarmCount[3  ] :=  AlarmCount[3]  + 1;   MpAlarmXSet(AlarmMpLink,'EventIDCode.2048');
		2049 :  AlarmCount[4  ] :=  AlarmCount[4]  + 1;   MpAlarmXSet(AlarmMpLink,'EventIDCode.2049');
		2050 :  AlarmCount[5  ] :=  AlarmCount[5]  + 1;   MpAlarmXSet(AlarmMpLink,'EventIDCode.2050');
		2051 :  AlarmCount[6  ] :=  AlarmCount[6]  + 1;   MpAlarmXSet(AlarmMpLink,'EventIDCode.2051');
		2052 :  AlarmCount[7  ] :=  AlarmCount[7]  + 1;   MpAlarmXSet(AlarmMpLink,'EventIDCode.2052');
		2053 :  AlarmCount[8  ] :=  AlarmCount[8]  + 1;   MpAlarmXSet(AlarmMpLink,'EventIDCode.2053');
		2054 :  AlarmCount[9  ] :=  AlarmCount[9]  + 1;   MpAlarmXSet(AlarmMpLink,'EventIDCode.2054');
		2055 :  AlarmCount[10 ] := AlarmCount[10]  + 1;   MpAlarmXSet(AlarmMpLink,'EventIDCode.2055');
		2056 :  AlarmCount[11 ] := AlarmCount[11]  + 1;   MpAlarmXSet(AlarmMpLink,'EventIDCode.2056');
		2057 :  AlarmCount[12 ] := AlarmCount[12]  + 1;   MpAlarmXSet(AlarmMpLink,'EventIDCode.2057');
		2058 :  AlarmCount[13 ] := AlarmCount[13]  + 1;   MpAlarmXSet(AlarmMpLink,'EventIDCode.2058');
		2060 :  AlarmCount[14 ] := AlarmCount[14]  + 1;   MpAlarmXSet(AlarmMpLink,'EventIDCode.2060');
		2061 :  AlarmCount[15 ] := AlarmCount[15]  + 1;   MpAlarmXSet(AlarmMpLink,'EventIDCode.2061');
		2063 :  AlarmCount[16 ] := AlarmCount[16]  + 1;   MpAlarmXSet(AlarmMpLink,'EventIDCode.2063');
		2064 :  AlarmCount[17 ] := AlarmCount[17]  + 1;   MpAlarmXSet(AlarmMpLink,'EventIDCode.2064');
		2066 :  AlarmCount[18 ] := AlarmCount[18]  + 1;   MpAlarmXSet(AlarmMpLink,'EventIDCode.2066');
		2067 :  AlarmCount[19 ] := AlarmCount[19]  + 1;   MpAlarmXSet(AlarmMpLink,'EventIDCode.2067');
		2068 :  AlarmCount[20 ] := AlarmCount[20]  + 1;   MpAlarmXSet(AlarmMpLink,'EventIDCode.2068');
		2069 :  AlarmCount[21 ] := AlarmCount[21]  + 1;   MpAlarmXSet(AlarmMpLink,'EventIDCode.2069');
		2070 :  AlarmCount[22 ] := AlarmCount[22]  + 1;   MpAlarmXSet(AlarmMpLink,'EventIDCode.2070');
		2071 :  AlarmCount[23 ] := AlarmCount[23]  + 1;   MpAlarmXSet(AlarmMpLink,'EventIDCode.2071');
		2074 :  AlarmCount[24 ] := AlarmCount[24]  + 1;   MpAlarmXSet(AlarmMpLink,'EventIDCode.2074');
		2077 :  AlarmCount[25 ] := AlarmCount[25]  + 1;   MpAlarmXSet(AlarmMpLink,'EventIDCode.2077');
		2080 :  AlarmCount[26 ] := AlarmCount[26]  + 1;   MpAlarmXSet(AlarmMpLink,'EventIDCode.7392');
		2082 :  AlarmCount[27 ] := AlarmCount[27]  + 1;   MpAlarmXSet(AlarmMpLink,'EventIDCode.2080');
		2083 :  AlarmCount[28 ] := AlarmCount[28]  + 1;   MpAlarmXSet(AlarmMpLink,'EventIDCode.2083');
		2084 :  AlarmCount[29 ] := AlarmCount[29]  + 1;   MpAlarmXSet(AlarmMpLink,'EventIDCode.2084');
		2085 :  AlarmCount[30 ] := AlarmCount[30]  + 1;   MpAlarmXSet(AlarmMpLink,'EventIDCode.2085');
		2090 :  AlarmCount[31 ] := AlarmCount[31]  + 1;   MpAlarmXSet(AlarmMpLink,'EventIDCode.2090');
		2091 :  AlarmCount[32 ] := AlarmCount[32]  + 1;   MpAlarmXSet(AlarmMpLink,'EventIDCode.2091');
		2092 :  AlarmCount[33 ] := AlarmCount[33]  + 1;   MpAlarmXSet(AlarmMpLink,'EventIDCode.2092');
		2093 :  AlarmCount[34 ] := AlarmCount[34]  + 1;   MpAlarmXSet(AlarmMpLink,'EventIDCode.2093');
		2094 :  AlarmCount[35 ] := AlarmCount[35]  + 1;   MpAlarmXSet(AlarmMpLink,'EventIDCode.2094');
		2095 :  AlarmCount[36 ] := AlarmCount[36]  + 1;   MpAlarmXSet(AlarmMpLink,'EventIDCode.2095');
		2097 :  AlarmCount[37 ] := AlarmCount[37]  + 1;   MpAlarmXSet(AlarmMpLink,'EventIDCode.2097');
		2098 :  AlarmCount[38 ] := AlarmCount[38]  + 1;   MpAlarmXSet(AlarmMpLink,'EventIDCode.2098');
		2099 :  AlarmCount[39 ] := AlarmCount[39]  + 1;   MpAlarmXSet(AlarmMpLink,'EventIDCode.2099');
		2100 :  AlarmCount[40 ] := AlarmCount[40]  + 1;   MpAlarmXSet(AlarmMpLink,'EventIDCode.2100');
		2101 :  AlarmCount[41 ] := AlarmCount[41]  + 1;   MpAlarmXSet(AlarmMpLink,'EventIDCode.2101');
		2102 :  AlarmCount[42 ] := AlarmCount[42]  + 1;   MpAlarmXSet(AlarmMpLink,'EventIDCode.2102');
		2103 :  AlarmCount[43 ] := AlarmCount[43]  + 1;   MpAlarmXSet(AlarmMpLink,'EventIDCode.2103');
		2104 :  AlarmCount[44 ] := AlarmCount[44]  + 1;   MpAlarmXSet(AlarmMpLink,'EventIDCode.2104');
		2105 :  AlarmCount[45 ] := AlarmCount[45]  + 1;   MpAlarmXSet(AlarmMpLink,'EventIDCode.2105');
		2106 :  AlarmCount[46 ] := AlarmCount[46]  + 1;   MpAlarmXSet(AlarmMpLink,'EventIDCode.2106');
		2107 :  AlarmCount[47 ] := AlarmCount[47]  + 1;   MpAlarmXSet(AlarmMpLink,'EventIDCode.2107');
		2108 :  AlarmCount[48 ] := AlarmCount[48]  + 1;   MpAlarmXSet(AlarmMpLink,'EventIDCode.2108');
		2109 :  AlarmCount[49 ] := AlarmCount[49]  + 1;   MpAlarmXSet(AlarmMpLink,'EventIDCode.2109');
		2110 :  AlarmCount[50 ] := AlarmCount[50]  + 1;   MpAlarmXSet(AlarmMpLink,'EventIDCode.2110');
		2111 :  AlarmCount[51 ] := AlarmCount[51]  + 1;   MpAlarmXSet(AlarmMpLink,'EventIDCode.2111');
		2112 :  AlarmCount[52 ] := AlarmCount[52]  + 1;   MpAlarmXSet(AlarmMpLink,'EventIDCode.2112');
		4096 :  AlarmCount[53 ] := AlarmCount[53]  + 1;   MpAlarmXSet(AlarmMpLink,'EventIDCode.4096');
		4097 :  AlarmCount[54 ] := AlarmCount[54]  + 1;   MpAlarmXSet(AlarmMpLink,'EventIDCode.4097');
		4101 :  AlarmCount[55 ] := AlarmCount[55]  + 1;   MpAlarmXSet(AlarmMpLink,'EventIDCode.4101');
		4102 :  AlarmCount[56 ] := AlarmCount[56]  + 1;   MpAlarmXSet(AlarmMpLink,'EventIDCode.4102');
		6144 :  AlarmCount[57 ] := AlarmCount[57]  + 1;   MpAlarmXSet(AlarmMpLink,'EventIDCode.6144');
		6165 :  AlarmCount[58 ] := AlarmCount[58]  + 1;   MpAlarmXSet(AlarmMpLink,'EventIDCode.6165');
		6148 :  AlarmCount[59 ] := AlarmCount[59]  + 1;   MpAlarmXSet(AlarmMpLink,'EventIDCode.6148');
		6149 :  AlarmCount[60 ] := AlarmCount[60]  + 1;   MpAlarmXSet(AlarmMpLink,'EventIDCode.6149');
		6156 :  AlarmCount[61 ] := AlarmCount[61]  + 1;   MpAlarmXSet(AlarmMpLink,'EventIDCode.6156');
		6157 :  AlarmCount[62 ] := AlarmCount[62]  + 1;   MpAlarmXSet(AlarmMpLink,'EventIDCode.6157');
		6158 :  AlarmCount[63 ] := AlarmCount[63]  + 1;   MpAlarmXSet(AlarmMpLink,'EventIDCode.6158');
		12288:  AlarmCount[64 ] := AlarmCount[64]  + 1;   MpAlarmXSet(AlarmMpLink,'EventIDCode.12288');
		12291:  AlarmCount[65 ] := AlarmCount[65]  + 1;   MpAlarmXSet(AlarmMpLink,'EventIDCode.12291');
		12293:  AlarmCount[66 ] := AlarmCount[66]  + 1;   MpAlarmXSet(AlarmMpLink,'EventIDCode.12293');
		12294:  AlarmCount[67 ] := AlarmCount[67]  + 1;   MpAlarmXSet(AlarmMpLink,'EventIDCode.12294');
		12295:  AlarmCount[68 ] := AlarmCount[68]  + 1;   MpAlarmXSet(AlarmMpLink,'EventIDCode.12295');
		12296:  AlarmCount[69 ] := AlarmCount[69]  + 1;   MpAlarmXSet(AlarmMpLink,'EventIDCode.12296');
		12297:  AlarmCount[70 ] := AlarmCount[70]  + 1;   MpAlarmXSet(AlarmMpLink,'EventIDCode.12297');
		12298:  AlarmCount[71 ] := AlarmCount[71]  + 1;   MpAlarmXSet(AlarmMpLink,'EventIDCode.12298');
		12299:  AlarmCount[72 ] := AlarmCount[72]  + 1;   MpAlarmXSet(AlarmMpLink,'EventIDCode.12299');
		12300:  AlarmCount[73 ] := AlarmCount[73]  + 1;   MpAlarmXSet(AlarmMpLink,'EventIDCode.12300');
		12301:  AlarmCount[74 ] := AlarmCount[74]  + 1;   MpAlarmXSet(AlarmMpLink,'EventIDCode.12301');
		12302:  AlarmCount[75 ] := AlarmCount[75]  + 1;   MpAlarmXSet(AlarmMpLink,'EventIDCode.12302');
		12303:  AlarmCount[76 ] := AlarmCount[76]  + 1;   MpAlarmXSet(AlarmMpLink,'EventIDCode.12303');
		12304:  AlarmCount[77 ] := AlarmCount[77]  + 1;   MpAlarmXSet(AlarmMpLink,'EventIDCode.12304');
		12305:  AlarmCount[78 ] := AlarmCount[78]  + 1;   MpAlarmXSet(AlarmMpLink,'EventIDCode.12305');
		12307:  AlarmCount[79 ] := AlarmCount[79]  + 1;   MpAlarmXSet(AlarmMpLink,'EventIDCode.12307');
		12312:  AlarmCount[80 ] := AlarmCount[80]  + 1;   MpAlarmXSet(AlarmMpLink,'EventIDCode.12312');
		12313:  AlarmCount[81 ] := AlarmCount[81]  + 1;   MpAlarmXSet(AlarmMpLink,'EventIDCode.12313');
		12314:  AlarmCount[82 ] := AlarmCount[82]  + 1;   MpAlarmXSet(AlarmMpLink,'EventIDCode.12314');
		12315:  AlarmCount[83 ] := AlarmCount[83]  + 1;   MpAlarmXSet(AlarmMpLink,'EventIDCode.12315');
		12316:  AlarmCount[84 ] := AlarmCount[84]  + 1;   MpAlarmXSet(AlarmMpLink,'EventIDCode.12316');
		12317:  AlarmCount[85 ] := AlarmCount[85]  + 1;   MpAlarmXSet(AlarmMpLink,'EventIDCode.12317');
		12320:  AlarmCount[86 ] := AlarmCount[86]  + 1;   MpAlarmXSet(AlarmMpLink,'EventIDCode.12320');
		12322:  AlarmCount[87 ] := AlarmCount[87]  + 1;   MpAlarmXSet(AlarmMpLink,'EventIDCode.12322');
		12323:  AlarmCount[88 ] := AlarmCount[88]  + 1;   MpAlarmXSet(AlarmMpLink,'EventIDCode.12323');
		12328:  AlarmCount[89 ] := AlarmCount[89]  + 1;   MpAlarmXSet(AlarmMpLink,'EventIDCode.12328');
		12330:  AlarmCount[90 ] := AlarmCount[90]  + 1;   MpAlarmXSet(AlarmMpLink,'EventIDCode.12330');
		12331:  AlarmCount[91 ] := AlarmCount[91]  + 1;   MpAlarmXSet(AlarmMpLink,'EventIDCode.12331');
		12333:  AlarmCount[92 ] := AlarmCount[92]  + 1;   MpAlarmXSet(AlarmMpLink,'EventIDCode.12333');
		12334:  AlarmCount[93 ] := AlarmCount[93]  + 1;   MpAlarmXSet(AlarmMpLink,'EventIDCode.12334');
		12335:  AlarmCount[94 ] := AlarmCount[94]  + 1;   MpAlarmXSet(AlarmMpLink,'EventIDCode.12335');
		12336:  AlarmCount[95 ] := AlarmCount[95]  + 1;   MpAlarmXSet(AlarmMpLink,'EventIDCode.12336');
		12337:  AlarmCount[96 ] := AlarmCount[96]  + 1;   MpAlarmXSet(AlarmMpLink,'EventIDCode.12337');
		12338:  AlarmCount[97 ] := AlarmCount[97]  + 1;   MpAlarmXSet(AlarmMpLink,'EventIDCode.12338');
		12340:  AlarmCount[98 ] := AlarmCount[98]  + 1;   MpAlarmXSet(AlarmMpLink,'EventIDCode.12340');
		12341:  AlarmCount[99 ] := AlarmCount[99]  + 1;   MpAlarmXSet(AlarmMpLink,'EventIDCode.12341');
		12342:  AlarmCount[100] := AlarmCount[100] + 1;   MpAlarmXSet(AlarmMpLink,'EventIDCode.12342');
		12343:  AlarmCount[101] := AlarmCount[101] + 1;   MpAlarmXSet(AlarmMpLink,'EventIDCode.12343');
		12344:  AlarmCount[102] := AlarmCount[102] + 1;   MpAlarmXSet(AlarmMpLink,'EventIDCode.12344');
		12345:  AlarmCount[103] := AlarmCount[103] + 1;   MpAlarmXSet(AlarmMpLink,'EventIDCode.12345');
		12346:  AlarmCount[104] := AlarmCount[104] + 1;   MpAlarmXSet(AlarmMpLink,'EventIDCode.12346');
		12347:  AlarmCount[105] := AlarmCount[105] + 1;   MpAlarmXSet(AlarmMpLink,'EventIDCode.12347');
		12348:  AlarmCount[106] := AlarmCount[106] + 1;   MpAlarmXSet(AlarmMpLink,'EventIDCode.12348');
		4007:   AlarmCount[107] := AlarmCount[107] + 1;   MpAlarmXSet(AlarmMpLink,'EventIDCode.4007');
		7230:   AlarmCount[108] := AlarmCount[108] + 1;   MpAlarmXSet(AlarmMpLink,'EventIDCode.7230');
		4005:   AlarmCount[109] := AlarmCount[109] + 1;   MpAlarmXSet(AlarmMpLink,'EventIDCode.4005');
		4098:   AlarmCount[110] := AlarmCount[110] + 1;   MpAlarmXSet(AlarmMpLink,'EventIDCode.4098');
		9106:   AlarmCount[111] := AlarmCount[111] + 1;   MpAlarmXSet(AlarmMpLink,'EventIDCode.9106');

		ELSE
			MpAlarmXSet(AlarmMpLink,'EventIDCode.xxxx');
		END_CASE

END_FUNCTION
```

### Program Logical/Source/SampleTrak/Diagnostic/SegTrace

#### Types.typ
```iecst
TYPE
	segTraceStateEnum :
		( (*State of Execution*)
		SEG_TRACE_IDLE, (*Idle State*)
		SEG_TRACE_READ_SEG, (*Read segment state, FB is being executed*)
		SEG_TRACE_CALC_RESULTS, (*Calculate any results from the parID being read*)
		SEG_TRACE_ADD_FAILS, (*Check for any failed segments state*)
		SEG_TRACE_DONE, (*Read/Check completed state*)
		SEG_TRACE_EXPORT, (*Export Trace results state*)
		SEG_TRACE_ERROR (*Error State*)
		);
END_TYPE
```

#### Variables.var
```iecst
VAR
	segTraceResults : ARRAY[0..MAX_SEGMENTS] OF segTraceResultsTyp;
	ProcessParId : MC_BR_SegProcessParID_AcpTrak;
	segIdx : USINT;
	i : USINT;
	state : segTraceStateEnum;
	RecipeXml : MpRecipeXml;
	RegPar : ARRAY[0..1] OF MpRecipeRegPar;
END_VAR
```

#### Cyclic.st
```iecst
PROGRAM _CYCLIC

	CASE state OF
		SEG_TRACE_IDLE:	//********************************************************************************************************* Trace Idle State
			IF gSegTraceIf.Cmds.Capture THEN
				gSegTraceIf.Status.Active := TRUE;
				gSegTraceIf.Status.Result := segTracePass;

				FOR i:=0 TO gSegTraceIf.Pars.SegmentCount - 1 DO
					brsmemset(ADR(segTraceResults[i].Values),0,SIZEOF(segTraceResults[i].Values));
					segTraceResults[i].BalancerPass := FALSE;
					segTraceResults[i].UDCActPass := FALSE;
					segTraceResults[i].UDCMiddlePass := FALSE;
					segTraceResults[i].BalancerSum := FALSE;
				END_FOR;
				brsmemset(ADR(gSegTraceIf.Status.Failures),0,SIZEOF(gSegTraceIf.Status.Failures));
				gSegTraceIf.Status.FailCount := 0;

				segIdx := 0;
				ProcessParId.Segment := ADR(TrackDiag.Seg[segIdx].SegmentLink) (*gSegTraceIf.Pars.Segments[segIdx]*);
				ProcessParId.Mode := mcACPTRAK_SEG_PARID_GET_NO_NCT;
				ProcessParId.NumberOfParIDs := 5;
				gSegTraceIf.Pars.ParIds[0].VariableAddress := ADR(segTraceResults[segIdx].Values.BalCurrent_Act_1);
				gSegTraceIf.Pars.ParIds[1].VariableAddress := ADR(segTraceResults[segIdx].Values.BalCurrent_Act_2);
				gSegTraceIf.Pars.ParIds[2].VariableAddress := ADR(segTraceResults[segIdx].Values.BalCurrent_Act_3);
				gSegTraceIf.Pars.ParIds[3].VariableAddress := ADR(segTraceResults[segIdx].Values.UdcAct);
				gSegTraceIf.Pars.ParIds[4].VariableAddress := ADR(segTraceResults[segIdx].Values.UdcMiddleAct);
				ProcessParId.DataAddress := ADR(gSegTraceIf.Pars.ParIds);
				ProcessParId.Execute := TRUE;

				//TODO: Validate that the gSegTraceIf.Pars.SegmentCount is < MAX_SEGMENTS

				state := SEG_TRACE_READ_SEG;
			ELSIF gSegTraceIf.Cmds.Export THEN
				RecipeXml.FileName := ADR(gSegTraceIf.Pars.Export.FileName);
				RecipeXml.Save := TRUE;

				state := SEG_TRACE_EXPORT;
			END_IF

		SEG_TRACE_READ_SEG://********************************************************************************************************* Trace Read Segment State
			IF ProcessParId.Error THEN
				gSegTraceIf.Status.Error := TRUE;
				gSegTraceIf.Status.Result := segTraceFail;
				state := SEG_TRACE_ERROR;
			ELSIF ProcessParId.Done THEN
				ProcessParId.Execute := FALSE;

				state := SEG_TRACE_CALC_RESULTS;
			END_IF
		SEG_TRACE_CALC_RESULTS://********************************************************************************************************* Trace Calculate Results State
			//Check the balancer sum
			segTraceResults[segIdx].BalancerSum := ABS(segTraceResults[segIdx].Values.BalCurrent_Act_1 + segTraceResults[segIdx].Values.BalCurrent_Act_2 + segTraceResults[segIdx].Values.BalCurrent_Act_3);
			IF segTraceResults[segIdx].BalancerSum > gSegTraceIf.Pars.BalancerCurrentLimit THEN
				gSegTraceIf.Status.Result := segTraceFail;
				segTraceResults[segIdx].BalancerPass := FALSE;
			ELSE
				segTraceResults[segIdx].BalancerPass := TRUE;
			END_IF
			//Check the UDC ACT vs power supply configured
			//TODO: Ideally the PS_UDC and POWERFAIL_DETECT_RATIO would be auto detected
			IF segTraceResults[segIdx].Values.UdcAct < gSegTraceIf.Pars.PS_UDC_Value * gSegTraceIf.Pars.PowerFailDetectRatio THEN
				gSegTraceIf.Status.Result := segTraceFail;
				segTraceResults[segIdx].UDCActPass := FALSE;
			ELSE
				segTraceResults[segIdx].UDCActPass := TRUE;
			END_IF

			//Check to verify UDC Middle is no more than +/- 7V around 1/2 UDC_ACT
			IF segTraceResults[segIdx].Values.UdcMiddleAct > segTraceResults[segIdx].Values.UdcAct / 2.0 + 7.0 OR segTraceResults[segIdx].Values.UdcMiddleAct < segTraceResults[segIdx].Values.UdcAct / 2.0 - 7.0 THEN
				gSegTraceIf.Status.Result := segTraceFail;
				segTraceResults[segIdx].UDCMiddlePass := FALSE;
			ELSE
				segTraceResults[segIdx].UDCMiddlePass := TRUE;
			END_IF

			segIdx := segIdx + 1;
			IF segIdx < gSegTraceIf.Pars.SegmentCount THEN
				ProcessParId.Segment :=  ADR(TrackDiag.Seg[segIdx].SegmentLink) (*gSegTraceIf.Pars.Segments[segIdx]*);
				gSegTraceIf.Pars.ParIds[0].VariableAddress := ADR(segTraceResults[segIdx].Values.BalCurrent_Act_1);
				gSegTraceIf.Pars.ParIds[1].VariableAddress := ADR(segTraceResults[segIdx].Values.BalCurrent_Act_2);
				gSegTraceIf.Pars.ParIds[2].VariableAddress := ADR(segTraceResults[segIdx].Values.BalCurrent_Act_3);
				gSegTraceIf.Pars.ParIds[3].VariableAddress := ADR(segTraceResults[segIdx].Values.UdcAct);
				gSegTraceIf.Pars.ParIds[4].VariableAddress := ADR(segTraceResults[segIdx].Values.UdcMiddleAct);
				ProcessParId.Execute := TRUE;

				state := SEG_TRACE_READ_SEG;

			ELSE
				state := SEG_TRACE_ADD_FAILS;
			END_IF
		SEG_TRACE_ADD_FAILS: //********************************************************************************************************* Trace Add Up Failures State
			FOR i := 0 TO gSegTraceIf.Pars.SegmentCount - 1 DO
				IF NOT segTraceResults[i].BalancerPass OR NOT segTraceResults[i].UDCActPass OR NOT segTraceResults[i].UDCMiddlePass THEN
					gSegTraceIf.Status.Failures[gSegTraceIf.Status.FailCount].SegName := TrackDiag.Seg[i].SegmentId; (*segTraceResults[i].SegmentName*)
					gSegTraceIf.Status.Failures[gSegTraceIf.Status.FailCount].WarningActive := TRUE;
					gSegTraceIf.Status.Failures[gSegTraceIf.Status.FailCount].BalancerFail := NOT segTraceResults[i].BalancerPass;
					gSegTraceIf.Status.Failures[gSegTraceIf.Status.FailCount].UDCActFail := NOT segTraceResults[i].UDCActPass;
					gSegTraceIf.Status.Failures[gSegTraceIf.Status.FailCount].UDCMiddleActFail := NOT segTraceResults[i].UDCMiddlePass;

					gSegTraceIf.Status.FailCount := gSegTraceIf.Status.FailCount + 1;
				END_IF
			END_FOR;

			IF gSegTraceIf.Status.FailCount > 0 THEN
				RecipeXml.FileName := ADR(gSegTraceIf.Pars.Export.FileName);
				RecipeXml.Save := TRUE;

				state := SEG_TRACE_EXPORT;
			ELSE
				gSegTraceIf.Status.Done := TRUE;

				state := SEG_TRACE_DONE;
			END_IF
		SEG_TRACE_DONE://********************************************************************************************************* Trace Done State
			IF NOT gSegTraceIf.Cmds.Capture THEN
				ProcessParId.Execute := FALSE;

				segIdx := 0;
				gSegTraceIf.Status.Active := FALSE;
				gSegTraceIf.Status.Done := FALSE;
				gSegTraceIf.Status.Error := FALSE;

				state := SEG_TRACE_IDLE;
			END_IF
		SEG_TRACE_EXPORT://********************************************************************************************************* Trace Export State
			IF RecipeXml.CommandDone THEN
				RecipeXml.Save := FALSE;
				IF gSegTraceIf.Cmds.Capture THEN
					gSegTraceIf.Status.Done := TRUE;
					state := SEG_TRACE_DONE;
				ELSE
					gSegTraceIf.Cmds.Export := FALSE;
					state := SEG_TRACE_IDLE;
				END_IF

			ELSIF RecipeXml.Error THEN
				state := SEG_TRACE_ERROR;
			END_IF
		SEG_TRACE_ERROR://********************************************************************************************************* Trace Error State
			IF gSegTraceIf.Cmds.ErrorReset THEN
				ProcessParId.Execute := FALSE;

				segIdx := 0;
				FOR i:=0 TO gSegTraceIf.Pars.SegmentCount - 1 DO
					brsmemset(ADR(segTraceResults[i].Values),0,SIZEOF(segTraceResults[i].Values));
					segTraceResults[i].BalancerPass := FALSE;
					segTraceResults[i].UDCActPass := FALSE;
					segTraceResults[i].UDCMiddlePass := FALSE;
					segTraceResults[i].BalancerSum := FALSE;
				END_FOR;
				brsmemset(ADR(gSegTraceIf.Status.Failures),0,SIZEOF(gSegTraceIf.Status.Failures));
				gSegTraceIf.Status.FailCount := 0;
				gSegTraceIf.Status.Active := FALSE;
				gSegTraceIf.Status.Done := FALSE;
				gSegTraceIf.Status.Error := FALSE;
				gSegTraceIf.Status.Result := segTraceUnknown;

				state := SEG_TRACE_IDLE;
			END_IF

	END_CASE;

	//FB Call
	ProcessParId();

	RecipeXml();
	RegPar[0]();
	RegPar[1]();
END_PROGRAM
```

#### Init.st
```iecst
PROGRAM _INIT
	//Setup the par ids we want to read
	gSegTraceIf.Pars.ParIds[0].DataType := mcACPTRAK_SEG_PARTYPE_REAL;
	gSegTraceIf.Pars.ParIds[0].ParID := 63801;	//Balancer current actual group 1

	gSegTraceIf.Pars.ParIds[1].DataType := mcACPTRAK_SEG_PARTYPE_REAL;
	gSegTraceIf.Pars.ParIds[1].ParID := 63802;	//Balancer current actual group 2

	gSegTraceIf.Pars.ParIds[2].DataType := mcACPTRAK_SEG_PARTYPE_REAL;
	gSegTraceIf.Pars.ParIds[2].ParID := 63803;	//Balancer current actual group 3

	gSegTraceIf.Pars.ParIds[3].DataType := mcACPTRAK_SEG_PARTYPE_REAL;
	gSegTraceIf.Pars.ParIds[3].ParID := mcACPPAR_UDC_ACT;	//Actual DC bus voltage value

	gSegTraceIf.Pars.ParIds[4].DataType := mcACPTRAK_SEG_PARTYPE_REAL;
	gSegTraceIf.Pars.ParIds[4].ParID := mcACPPAR_UDC_MIDDLE_ACT;	//Actual mid point DC bus voltage value

	//Setup the interface as needed
	gSegTraceIf.Pars.BalancerCurrentLimit := 24;
	gSegTraceIf.Pars.PS_UDC_Value := 58;
	gSegTraceIf.Pars.PowerFailDetectRatio := 0.779;

	//Setup the MpRecipe Blocks
	IF DiagCpuIsSimulated() THEN
		gSegTraceIf.Pars.Export.FileDev := 'SegTraceSim';
	ELSE
		gSegTraceIf.Pars.Export.FileDev := 'SegTrace';
	END_IF
	gSegTraceIf.Pars.Export.FileName := 'DefaultSegTraceExport';
	RecipeXml.MpLink := ADR(gMpRecipeDiagXml);
	RecipeXml.Enable := TRUE;
	RecipeXml.Category := ADR('SegTrace');
	RecipeXml.DeviceName := ADR(gSegTraceIf.Pars.Export.FileDev);
	RegPar[0].Enable := TRUE;
	RegPar[0].Category := ADR('SegTrace');
	RegPar[0].MpLink := ADR(gMpRecipeDiagXml);
	RegPar[0].PVName := ADR('gSegTraceIf.Status');
	RegPar[1].Enable := TRUE;
	RegPar[1].Category := ADR('SegTrace');
	RegPar[1].MpLink := ADR(gMpRecipeDiagXml);
	RegPar[1].PVName := ADR('SegTrace:segTraceResults');

	gSegTraceIf.Pars.SegmentCount := TrackDiag.SegmentCount;

	//FB Call
	RecipeXml();
	RegPar[0]();
	RegPar[1]();
END_PROGRAM
```

### Program Logical/Source/SampleTrak/Diagnostic/TrackMap

#### Variables.var
```iecst
VAR
	paperCore : TrkPaperCore;
	Offset : UDINT;
	clickId : STRING[160];
	i : INT;
	clickedSegment : TrkPaperCoreSegmentType;
	SegIndex : INT;
END_VAR
```

#### Cyclic.st
```iecst
PROGRAM _CYCLIC

	paperCore();

	clickId;

	// compare the elementID clicked on in paper with the configured ID to find and set the array index for the list binding
	FOR SegIndex:= 0 TO NUM_SEG DO

		IF TrackDiag.Seg.SegList[SegIndex].Name = DELETE(clickId,1,1) THEN // clickId contains a leading # which needs to be removed

			clickedSegment := TrackDiag.Seg.SegList[SegIndex];
			EXIT;
		END_IF

	END_FOR

END_PROGRAM
```

#### Init.st
```iecst
PROGRAM _INIT

	paperCore.SegmentCount := TrackDiag.Seg.SegCount;

	paperCore.Segments := ADR(TrackDiag.Seg.SegList);

	paperCore.Options := ADR(paperOptions);

	paperCore.Enable := TRUE;

END_PROGRAM
```

### Program Logical/Source/SampleTrak/Diagnostic/TrakLogger (IEC)

#### Main.st - Init, cyclic, exit code
```iecst
//////////////////////////////////////////////////////////////////////////////////////////////////////////////////////////////
//
// Copyright B&R Industrial Automation GmbH
// Author    B&R
// Created   Feb 1, 2018
//
// trak motion logger filter task (optional)
// TC#8 => mandatory to be attached to idle task class!
//
// * filters the "Motion" logger to display the newest 10 entries with severity "Error" or "Warning" entered by segments
//
// "TrakLogger" - local interface structure
//
//////////////////////////////////////////////////////////////////////////////////////////////////////////////////////////////

PROGRAM _CYCLIC

	MC_BR_AsmReadStatus_AcpTrak_0.Assembly := TrakLogger.AssemblyRef;
	MC_BR_AsmReadStatus_AcpTrak_0.Enable := TRUE;
	MC_BR_AsmReadStatus_AcpTrak_0();

	MC_BR_SegCommandError_AcpTrak_0(Segment := ADR(TrackDiag.Seg.SegList[0].McType));

	IF MC_BR_SegCommandError_AcpTrak_0.Done THEN
		MC_BR_SegCommandError_AcpTrak_0.Execute := FALSE;
	END_IF

	IF EDGEPOS(MC_BR_AsmReadStatus_AcpTrak_0.AssemblyErrorStop) THEN
		TrakLogger.CmdRefresh := TRUE;
	END_IF

	REPEAT
		StepLast := Step;

		CASE Step OF

			//////////////////////////////////////////////////////////////////////////////////////////////////////////////////////////////
			// command
			TRAK_COMMAND:
				IF TrakLogger.CmdRefresh THEN
					Step := TRAK_RESET;
				END_IF

			//////////////////////////////////////////////////////////////////////////////////////////////////////////////////////////////
			// wait till all messages are entered into logger
			TRAK_RESET:
				FubTonWaitFirst.IN := TRUE;
				FubTonWaitFirst.PT := T#1s;
				FubTonWaitFirst();
				IF FubTonWaitFirst.Q THEN
					FubTonWaitFirst.IN := FALSE;

					brsmemset(ADR(TrakLogger.Record), 0, SIZEOF(TrakLogger.Record));
					TrakLogger.Message := '';
					SegmentErrorFound := 0;

					brsmemset(ADR(AlarmCount), 0, SIZEOF(AlarmCount));

					ArEventLogGetIdent_0.Execute			:= FALSE;
					ArEventLogGetLatestRecordID_0.Execute	:= FALSE;
					ArEventLogGetPreviousRecordID_0.Execute	:= FALSE;
					ArEventLogRead_0.Execute				:= FALSE;
					ArEventLogReadObjectID_0.Execute		:= FALSE;
					ArEventLogReadDescription_0.Execute		:= FALSE;
					Step := TRAK_GET_IDENT;
				END_IF

			///////////////////////////////////////////////////////////////////////////
			// open logger and read first EventID
			TRAK_GET_IDENT:
				ArEventLogGetIdent_0.Execute	:= TRUE;
				brsstrcpy(ADR(ArEventLogGetIdent_0.Name), ADR('$$motion'));
				Step := TRAK_GET_IDENT_WAIT;

			TRAK_GET_IDENT_WAIT:
				IF ArEventLogGetIdent_0.Done THEN
					Ident := ArEventLogGetIdent_0.Ident;
					ArEventLogGetIdent_0.Execute := FALSE;
					Step := TRAK_GET_LATEST_ID;
				ELSIF ArEventLogGetIdent_0.Error THEN
					TrakLogger.Message := 'Error GetIdent';
					Step := TRAK_ERROR;
				END_IF

			TRAK_GET_LATEST_ID:
				ArEventLogGetLatestRecordID_0.Execute	:= TRUE;
				ArEventLogGetLatestRecordID_0.Ident		:= Ident;
				Step := TRAK_GET_LATEST_ID_WAIT;

			TRAK_GET_LATEST_ID_WAIT:
				IF ArEventLogGetLatestRecordID_0.Done THEN
					RecordID := ArEventLogGetLatestRecordID_0.RecordID;
					ArEventLogGetLatestRecordID_0.Execute := FALSE;
					Step := TRAK_READ_ID;
				ELSIF ArEventLogGetLatestRecordID_0.Error THEN
					TrakLogger.Message := 'Error GetLatestRecordID';
					Step := TRAK_ERROR;
				END_IF

			///////////////////////////////////////////////////////////////////////////
			// read previous EventID
			TRAK_GET_PREVIOUS_ID:
				ArEventLogGetPreviousRecordID_0.Execute		:= TRUE;
				ArEventLogGetPreviousRecordID_0.Ident		:= Ident;
				ArEventLogGetPreviousRecordID_0.RecordID	:= RecordID;
				Step := TRAK_GET_PREVIOUS_ID_WAIT;

			TRAK_GET_PREVIOUS_ID_WAIT:
				IF ArEventLogGetPreviousRecordID_0.Done THEN
					RecordID := ArEventLogGetPreviousRecordID_0.PrevRecordID;
					ArEventLogGetPreviousRecordID_0.Execute := FALSE;
					Step := TRAK_READ_ID;
				ELSIF ArEventLogGetPreviousRecordID_0.Error THEN
					IF ArEventLogGetPreviousRecordID_0.StatusID = arEVENTLOG_ERR_RECORDID_INVALID THEN		// reached end of logger
						ArEventLogGetPreviousRecordID_0.Execute := FALSE;
						Step := TRAK_DONE;
					ELSE
						TrakLogger.Message := 'Error GetPreviousRecordID';
						Step := TRAK_ERROR;
					END_IF
				END_IF

			///////////////////////////////////////////////////////////////////////////
			// check if severity is 'Error' or 'Warning'
			TRAK_READ_ID:
				ArEventLogRead_0.Execute	:= TRUE;
				ArEventLogRead_0.Ident		:= Ident;
				ArEventLogRead_0.RecordID	:= RecordID;
				Step := TRAK_READ_ID_WAIT;

			TRAK_READ_ID_WAIT:
				IF ArEventLogRead_0.Done THEN
					EventID := ArEventLogRead_0.EventID;
					ArEventLogRead_0.Execute := FALSE;
					EventTimeStamp := ArEventLogRead_0.TimeStamp;

					EventIDSeverity	:= DINT_TO_USINT(SHR(EventID, 30) AND 16#03);
					EventIDFacility	:= DINT_TO_UINT(SHR(EventID, 16) AND 16#0FFF);
					EventIDCode		:= DINT_TO_UINT(SHR(EventID, 0) AND 16#FFFF);

					IF ((EventIDSeverity = arEVENTLOG_SEVERITY_ERROR) AND (TrakLogger.ParaShowSegError)) THEN
						Step := TRAK_CHECK_FILTER;
					ELSIF ((EventIDSeverity = arEVENTLOG_SEVERITY_WARNING) AND (TrakLogger.ParaShowSegWarning)) THEN
						Step := TRAK_CHECK_FILTER;
					ELSE
						Step := TRAK_GET_PREVIOUS_ID;
					END_IF
				ELSIF ArEventLogRead_0.Error THEN
					TrakLogger.Message := 'Error ReadRecordID';
					Step := TRAK_ERROR;
				END_IF

			///////////////////////////////////////////////////////////////////////////
			// check if 'Error' has been entered by a Segment
			TRAK_CHECK_FILTER:
				ArEventLogReadObjectID_0.Execute	:= TRUE;
				ArEventLogReadObjectID_0.Ident		:= Ident;
				ArEventLogReadObjectID_0.RecordID	:= RecordID;
				Step := TRAK_CHECK_FILTER_WAIT;

			TRAK_CHECK_FILTER_WAIT:
				IF ArEventLogReadObjectID_0.Done THEN
					ObjectID := ArEventLogReadObjectID_0.ObjectID;
					ArEventLogReadObjectID_0.Execute := FALSE;
					IF brsmemcmp(ADR(ObjectID), ADR(TrakLogger.ParaSegFilter), 3) = 0 THEN
						Step := TRAK_READ_DESCRIPTION;
					ELSE
						Step := TRAK_GET_PREVIOUS_ID;
					END_IF
				ELSIF ArEventLogReadObjectID_0.Error THEN
					TrakLogger.Message := 'Error ReadObjectID';
					Step := TRAK_ERROR;
				END_IF

			///////////////////////////////////////////////////////////////////////////
			// read and display description text if filter criterias are matching
			TRAK_READ_DESCRIPTION:
				ArEventLogReadDescription_0.Execute			:= TRUE;
				ArEventLogReadDescription_0.Ident			:= Ident;
				ArEventLogReadDescription_0.RecordID		:= RecordID;
			//	ArEventLogReadDescription_0.LanguageCode	:= ;
			//	ArEventLogReadDescription_0.Qualifier		:= ;
				ArEventLogReadDescription_0.TextBuffer		:= ADR(Description);
				ArEventLogReadDescription_0.TextBufferSize	:= SIZEOF(Description);
				Step := TRAK_READ_DESCRIPTION_WAIT;

			TRAK_READ_DESCRIPTION_WAIT:
				IF ArEventLogReadDescription_0.Done THEN
					ArEventLogReadDescription_0.Execute := FALSE;
					Step := TRAK_UPDATE_LIST;
				ELSIF ArEventLogReadDescription_0.Error THEN
					TrakLogger.Message := 'Error ReadDescription';
					Step := TRAK_ERROR;
				END_IF

			TRAK_UPDATE_LIST:
				TrakLogger.Record[SegmentErrorFound].ObjectID			:= ObjectID;
				TrakLogger.Record[SegmentErrorFound].EventID			:= EventID;
				TrakLogger.Record[SegmentErrorFound].EventIDSeverity	:= EventIDSeverity;
				TrakLogger.Record[SegmentErrorFound].EventIDFacility	:= EventIDFacility;
				TrakLogger.Record[SegmentErrorFound].EventIDCode		:= EventIDCode;
				TrakLogger.Record[SegmentErrorFound].Description		:= Description;

				TrakLogger.Record[SegmentErrorFound].EventTimeStamp	:= UDINT_TO_TIME((EventTimeStamp.sec MOD (24*60*60))*1000 + (EventTimeStamp.nsec / 1000000));		// convert to TIME format (ms since start of day)

				brsstrcpy(ADR(TrakLogger.Record[SegmentErrorFound].Text), ADR(''));
				ascTIME(TrakLogger.Record[SegmentErrorFound].EventTimeStamp, ADR(TempString), SIZEOF(TempString));
				TIME_TO_TIMEStructure(TrakLogger.Record[SegmentErrorFound].EventTimeStamp,ADR(TimeStruct)); // for checking against older entries

				brsstrcat(ADR(TrakLogger.Record[SegmentErrorFound].Text), ADR(TempString));
				brsstrcat(ADR(TrakLogger.Record[SegmentErrorFound].Text), ADR(' => '));

				brsstrcat(ADR(TrakLogger.Record[SegmentErrorFound].Text), ADR(ObjectID));

				brsstrcat(ADR(TrakLogger.Record[SegmentErrorFound].Text), ADR(': Error '));
				brsitoa(EventIDCode, ADR(TempString));
				brsstrcat(ADR(TrakLogger.Record[SegmentErrorFound].Text), ADR(TempString));

				brsstrcat(ADR(TrakLogger.Record[SegmentErrorFound].Text), ADR(' => '));
				brsstrcat(ADR(TrakLogger.Record[SegmentErrorFound].Text), ADR(Description));

				IF SegmentErrorFound = 0 THEN
					FirstEntryCheckSum := TimeStruct.minute; // save the timestamp minute of the first entry as checksum
				END_IF

				SegmentErrorFound := SegmentErrorFound + 1;

				SetAlarmIDCode; //case statement to trigger alarms

				// stop reading the logger when the end of the array is reached OR
				// when the entries start having a different timestamp which means they are older
				IF SegmentErrorFound > 499 OR (FirstEntryCheckSum <> (TimeStruct.minute) ) THEN
					Step := TRAK_DONE;
				ELSE
					Step := TRAK_GET_PREVIOUS_ID;
				END_IF

			//////////////////////////////////////////////////////////////////////////////////////////////////////////////////////////////
			TRAK_DONE:
				TrakLogger.CmdRefresh := FALSE;
				Step := TRAK_COMMAND;

			//////////////////////////////////////////////////////////////////////////////////////////////////////////////////////////////
			TRAK_ERROR:
				IF TrakLogger.CmdRefresh = 0 THEN
					TrakLogger.Message := '';
					ArEventLogGetIdent_0.Execute			:= FALSE;
					ArEventLogGetLatestRecordID_0.Execute	:= FALSE;
					ArEventLogGetPreviousRecordID_0.Execute	:= FALSE;
					ArEventLogRead_0.Execute				:= FALSE;
					ArEventLogReadObjectID_0.Execute		:= FALSE;
					ArEventLogReadDescription_0.Execute		:= FALSE;
					Step := TRAK_COMMAND;
				END_IF

		END_CASE

		ArEventLogGetIdent_0();
		ArEventLogGetLatestRecordID_0();
		ArEventLogGetPreviousRecordID_0();
		ArEventLogRead_0();
		ArEventLogReadObjectID_0();
		ArEventLogReadDescription_0();

	UNTIL
		// to speed processing time of this sequence up: repeat sequence till the step is not changing any more (sequence is waiting for a FUB)
		Step = StepLast

	END_REPEAT

END_PROGRAM

PROGRAM _EXIT

END_PROGRAM
```

#### Init.st - Init, cyclic, exit code
```iecst
//////////////////////////////////////////////////////////////////////////////////////////////////////////////////////////////
//
// Copyright B&R Industrial Automation GmbH
// Author    B&R
// Created   Feb 1, 2018
//
// trak motion logger filter task (optional)
// TC#8 => mandatory to be attached to idle task class!
//
// * filters the "Motion" logger to display the newest 10 entries with severity "Error" or "Warning" entered by segments
//
// "TrakLogger" - local interface structure
//
//////////////////////////////////////////////////////////////////////////////////////////////////////////////////////////////

PROGRAM _INIT

	TrakLogger.AssemblyRef			:= ADR(DiagInterface.SampleTrak);
	TrakLogger.CmdRefresh			:= FALSE;
	TrakLogger.ParaShowSegError		:= TRUE;
	TrakLogger.ParaShowSegWarning	:= TRUE;
	TrakLogger.ParaSegFilter		:= 'gSeg_';

	Step := TRAK_COMMAND;

END_PROGRAM
```

#### Types.typ - Local data types
```iecst
(*read & filter motion logger*)

TYPE
	TrakLoggerType : 	STRUCT
		AssemblyRef : REFERENCE TO McAssemblyType; (*assembly reference - ADR(gAssembly_1)*)
		CmdRefresh : BOOL; (*command read & filter motion logger*)
		ParaShowSegError : BOOL; (*filter - show motion logger enties severity error*)
		ParaShowSegWarning : BOOL; (*filter - show motion logger enties severity warning*)
		ParaSegFilter : STRING[8]; (*show only entries with names beginning with this string*)
		Message : STRING[256]; (*message ArEventLog handling*)
		Record : ARRAY[0..500]OF TrakLoggerRecordType;
	END_STRUCT;
	TrakLoggerRecordType : 	STRUCT
		ObjectID : STRING[36]; (*logger entry "Entered by"*)
		EventID : DINT; (*logger entry "ID"*)
		EventIDSeverity : USINT; (*logger entry "Severity"*)
		EventIDFacility : UINT; (*logger entry "Facility"*)
		EventIDCode : UINT; (*logger entry "Code"*)
		EventTimeStamp : TIME; (*logger entry "Time"*)
		Text : STRING[300]; (*logger entry "Description"*)
		Description : STRING[256]; (*logger entry "Description"*)
	END_STRUCT;
END_TYPE

(*enum*)

TYPE
	StepEnum :
		(
		TRAK_COMMAND := 0,
		TRAK_RESET,
		TRAK_GET_IDENT := 10,
		TRAK_GET_IDENT_WAIT,
		TRAK_GET_LATEST_ID,
		TRAK_GET_LATEST_ID_WAIT,
		TRAK_GET_PREVIOUS_ID := 20,
		TRAK_GET_PREVIOUS_ID_WAIT,
		TRAK_READ_ID := 30,
		TRAK_READ_ID_WAIT,
		TRAK_CHECK_FILTER := 40,
		TRAK_CHECK_FILTER_WAIT,
		TRAK_READ_DESCRIPTION := 50,
		TRAK_READ_DESCRIPTION_WAIT,
		TRAK_UPDATE_LIST := 60,
		TRAK_DONE := 90,
		TRAK_ERROR := 99
		);
END_TYPE
```

#### Variables.var - Local variables
```iecst
(*read & filter motion logger*)
VAR
	TrakLogger : TrakLoggerType;
	Step : StepEnum := (0);
	StepLast : StepEnum := (0);
	Ident : ArEventLogIdentType := (0);
	RecordID : ArEventLogRecordIDType := (0);
	EventTimeStamp : ArEventLogTimeStampType := (0);
	EventID : DINT := 0;
	EventIDSeverity : USINT := 0;
	EventIDFacility : UINT := 0;
	EventIDCode : UINT := 0;
	ObjectID : STRING[36] := '';
	Description : STRING[256] := '';
	TempString : STRING[32] := '';
	SegmentErrorFound : USINT := 0;
END_VAR
(*assembly FUB*)
VAR
	MC_BR_AsmReadStatus_AcpTrak_0 : MC_BR_AsmReadStatus_AcpTrak;
END_VAR
(*ArEventLog FUB*)
VAR
	FubTonWaitFirst : TON := (0);
	ArEventLogGetIdent_0 : ArEventLogGetIdent := (0);
	ArEventLogGetLatestRecordID_0 : ArEventLogGetLatestRecordID := (0);
	ArEventLogGetPreviousRecordID_0 : ArEventLogGetPreviousRecordID := (0);
	ArEventLogRead_0 : ArEventLogRead := (0);
	ArEventLogReadObjectID_0 : ArEventLogReadObjectID := (0);
	ArEventLogReadDescription_0 : ArEventLogReadDescription := (0);
	MC_BR_SegCommandError_AcpTrak_0 : MC_BR_SegCommandError_AcpTrak;
	AlarmCount : ARRAY[0..119] OF UDINT;
	TimeStruct : TIMEStructure;
	FirstEntryCheckSum : USINT;
END_VAR
```

#### Action.st
```iecst
ACTION SetAlarmIDCode:

		// EventIDCode add new alarms triggers at the end otherwise
		// the AlarmCount has to be adjusted not just here but also for all the alarms in the MpAlarmX config

		CASE EventIDCode OF
		// every time the alarm is triggered it's counted so a total count can be displayed in the alarm message
		1	 : AlarmCount[0] := AlarmCount[0] + 1;   MpAlarmXSet(DiagInterface.AlarmCore,'EventIDCode.1	');
		2	 : AlarmCount[1] := AlarmCount[1] + 1;   MpAlarmXSet(DiagInterface.AlarmCore,'EventIDCode.2	');
		7	 : AlarmCount[2] := AlarmCount[2] + 1;   MpAlarmXSet(DiagInterface.AlarmCore,'EventIDCode.7	');
		2048 : AlarmCount[3] := AlarmCount[3] + 1;   MpAlarmXSet(DiagInterface.AlarmCore,'EventIDCode.2048');
		2049 : AlarmCount[4] := AlarmCount[4] + 1;   MpAlarmXSet(DiagInterface.AlarmCore,'EventIDCode.2049');
		2050 : AlarmCount[5] := AlarmCount[5] + 1;   MpAlarmXSet(DiagInterface.AlarmCore,'EventIDCode.2050');
		2051 : AlarmCount[6] := AlarmCount[6] + 1;   MpAlarmXSet(DiagInterface.AlarmCore,'EventIDCode.2051');
		2052 : AlarmCount[7] := AlarmCount[7] + 1;   MpAlarmXSet(DiagInterface.AlarmCore,'EventIDCode.2052');
		2053 : AlarmCount[8] := AlarmCount[8] + 1;   MpAlarmXSet(DiagInterface.AlarmCore,'EventIDCode.2053');
		2054 : AlarmCount[9] := AlarmCount[9] + 1;   MpAlarmXSet(DiagInterface.AlarmCore,'EventIDCode.2054');
		2055 : AlarmCount[10] := AlarmCount[10] + 1; MpAlarmXSet(DiagInterface.AlarmCore,'EventIDCode.2055');
		2056 : AlarmCount[11] := AlarmCount[11] + 1; MpAlarmXSet(DiagInterface.AlarmCore,'EventIDCode.2056');
		2057 : AlarmCount[12] := AlarmCount[12] + 1; MpAlarmXSet(DiagInterface.AlarmCore,'EventIDCode.2057');
		2058 : AlarmCount[13] := AlarmCount[13] + 1; MpAlarmXSet(DiagInterface.AlarmCore,'EventIDCode.2058');
		2060 : AlarmCount[14] := AlarmCount[14] + 1; MpAlarmXSet(DiagInterface.AlarmCore,'EventIDCode.2060');
		2061 : AlarmCount[15] := AlarmCount[15] + 1; MpAlarmXSet(DiagInterface.AlarmCore,'EventIDCode.2061');
		2063 : AlarmCount[16] := AlarmCount[16] + 1; MpAlarmXSet(DiagInterface.AlarmCore,'EventIDCode.2063');
		2064 : AlarmCount[17] := AlarmCount[17] + 1; MpAlarmXSet(DiagInterface.AlarmCore,'EventIDCode.2064');
		2066 : AlarmCount[18] := AlarmCount[18] + 1; MpAlarmXSet(DiagInterface.AlarmCore,'EventIDCode.2066');
		2067 : AlarmCount[19] := AlarmCount[19] + 1; MpAlarmXSet(DiagInterface.AlarmCore,'EventIDCode.2067');
		2068 : AlarmCount[20] := AlarmCount[20] + 1; MpAlarmXSet(DiagInterface.AlarmCore,'EventIDCode.2068');
		2069 : AlarmCount[21] := AlarmCount[21] + 1; MpAlarmXSet(DiagInterface.AlarmCore,'EventIDCode.2069');
		2070 : AlarmCount[22] := AlarmCount[22] + 1; MpAlarmXSet(DiagInterface.AlarmCore,'EventIDCode.2070');
		2071 : AlarmCount[23] := AlarmCount[23] + 1; MpAlarmXSet(DiagInterface.AlarmCore,'EventIDCode.2071');
		2074 : AlarmCount[24] := AlarmCount[24] + 1; MpAlarmXSet(DiagInterface.AlarmCore,'EventIDCode.2074');
		2077 : AlarmCount[25] := AlarmCount[25] + 1; MpAlarmXSet(DiagInterface.AlarmCore,'EventIDCode.2077');
		2080 : AlarmCount[26] := AlarmCount[26] + 1; MpAlarmXSet(DiagInterface.AlarmCore,'EventIDCode.7392');
		2082 : AlarmCount[27] := AlarmCount[27] + 1; MpAlarmXSet(DiagInterface.AlarmCore,'EventIDCode.2080');
		2083 : AlarmCount[28] := AlarmCount[28] + 1; MpAlarmXSet(DiagInterface.AlarmCore,'EventIDCode.2083');
		2084 : AlarmCount[29] := AlarmCount[29] + 1; MpAlarmXSet(DiagInterface.AlarmCore,'EventIDCode.2084');
		2085 : AlarmCount[30] := AlarmCount[30] + 1; MpAlarmXSet(DiagInterface.AlarmCore,'EventIDCode.2085');
		2090 : AlarmCount[31] := AlarmCount[31] + 1; MpAlarmXSet(DiagInterface.AlarmCore,'EventIDCode.2090');
		2091 : AlarmCount[32] := AlarmCount[32] + 1; MpAlarmXSet(DiagInterface.AlarmCore,'EventIDCode.2091');
		2092 : AlarmCount[33] := AlarmCount[33] + 1; MpAlarmXSet(DiagInterface.AlarmCore,'EventIDCode.2092');
		2093 : AlarmCount[34] := AlarmCount[34] + 1; MpAlarmXSet(DiagInterface.AlarmCore,'EventIDCode.2093');
		2094 : AlarmCount[35] := AlarmCount[35] + 1; MpAlarmXSet(DiagInterface.AlarmCore,'EventIDCode.2094');
		2095 : AlarmCount[36] := AlarmCount[36] + 1; MpAlarmXSet(DiagInterface.AlarmCore,'EventIDCode.2095');
		2097 : AlarmCount[37] := AlarmCount[37] + 1; MpAlarmXSet(DiagInterface.AlarmCore,'EventIDCode.2097');
		2098 : AlarmCount[38] := AlarmCount[38] + 1; MpAlarmXSet(DiagInterface.AlarmCore,'EventIDCode.2098');
		2099 : AlarmCount[39] := AlarmCount[39] + 1; MpAlarmXSet(DiagInterface.AlarmCore,'EventIDCode.2099');
		2100 : AlarmCount[40] := AlarmCount[40] + 1; MpAlarmXSet(DiagInterface.AlarmCore,'EventIDCode.2100');
		2101 : AlarmCount[41] := AlarmCount[41] + 1; MpAlarmXSet(DiagInterface.AlarmCore,'EventIDCode.2101');
		2102 : AlarmCount[42] := AlarmCount[42] + 1; MpAlarmXSet(DiagInterface.AlarmCore,'EventIDCode.2102');
		2103 : AlarmCount[43] := AlarmCount[43] + 1; MpAlarmXSet(DiagInterface.AlarmCore,'EventIDCode.2103');
		2104 : AlarmCount[44] := AlarmCount[44] + 1; MpAlarmXSet(DiagInterface.AlarmCore,'EventIDCode.2104');
		2105 : AlarmCount[45] := AlarmCount[45] + 1; MpAlarmXSet(DiagInterface.AlarmCore,'EventIDCode.2105');
		2106 : AlarmCount[46] := AlarmCount[46] + 1; MpAlarmXSet(DiagInterface.AlarmCore,'EventIDCode.2106');
		2107 : AlarmCount[47] := AlarmCount[47] + 1; MpAlarmXSet(DiagInterface.AlarmCore,'EventIDCode.2107');
		2108 : AlarmCount[48] := AlarmCount[48] + 1; MpAlarmXSet(DiagInterface.AlarmCore,'EventIDCode.2108');
		2109 : AlarmCount[49] := AlarmCount[49] + 1; MpAlarmXSet(DiagInterface.AlarmCore,'EventIDCode.2109');
		2110 : AlarmCount[50] := AlarmCount[50] + 1; MpAlarmXSet(DiagInterface.AlarmCore,'EventIDCode.2110');
		2111 : AlarmCount[51] := AlarmCount[51] + 1; MpAlarmXSet(DiagInterface.AlarmCore,'EventIDCode.2111');
		2112 : AlarmCount[52] := AlarmCount[52] + 1; MpAlarmXSet(DiagInterface.AlarmCore,'EventIDCode.2112');
		4096 : AlarmCount[53] := AlarmCount[53] + 1; MpAlarmXSet(DiagInterface.AlarmCore,'EventIDCode.4096');
		4097 : AlarmCount[54] := AlarmCount[54] + 1; MpAlarmXSet(DiagInterface.AlarmCore,'EventIDCode.4097');
		4101 : AlarmCount[55] := AlarmCount[55] + 1; MpAlarmXSet(DiagInterface.AlarmCore,'EventIDCode.4101');
		4102 : AlarmCount[56] := AlarmCount[56] + 1; MpAlarmXSet(DiagInterface.AlarmCore,'EventIDCode.4102');
		6144 : AlarmCount[57] := AlarmCount[57] + 1; MpAlarmXSet(DiagInterface.AlarmCore,'EventIDCode.6144');
		6165 : AlarmCount[58] := AlarmCount[58] + 1; MpAlarmXSet(DiagInterface.AlarmCore,'EventIDCode.6165');
		6148 : AlarmCount[59] := AlarmCount[59] + 1; MpAlarmXSet(DiagInterface.AlarmCore,'EventIDCode.6148');
		6149 : AlarmCount[60] := AlarmCount[60] + 1; MpAlarmXSet(DiagInterface.AlarmCore,'EventIDCode.6149');
		6156 : AlarmCount[61] := AlarmCount[61] + 1; MpAlarmXSet(DiagInterface.AlarmCore,'EventIDCode.6156');
		6157 : AlarmCount[62] := AlarmCount[62] + 1; MpAlarmXSet(DiagInterface.AlarmCore,'EventIDCode.6157');
		6158 : AlarmCount[63] := AlarmCount[63] + 1; MpAlarmXSet(DiagInterface.AlarmCore,'EventIDCode.6158');
		12288:  AlarmCount[64] := AlarmCount[64] + 1; MpAlarmXSet(DiagInterface.AlarmCore,'EventIDCode.12288');
		12291:  AlarmCount[65] := AlarmCount[65] + 1; MpAlarmXSet(DiagInterface.AlarmCore,'EventIDCode.12291');
		12293:  AlarmCount[66] := AlarmCount[66] + 1; MpAlarmXSet(DiagInterface.AlarmCore,'EventIDCode.12293');
		12294:  AlarmCount[67] := AlarmCount[67] + 1; MpAlarmXSet(DiagInterface.AlarmCore,'EventIDCode.12294');
		12295:  AlarmCount[68] := AlarmCount[68] + 1; MpAlarmXSet(DiagInterface.AlarmCore,'EventIDCode.12295');
		12296:  AlarmCount[69] := AlarmCount[69] + 1; MpAlarmXSet(DiagInterface.AlarmCore,'EventIDCode.12296');
		12297:  AlarmCount[70] := AlarmCount[70] + 1; MpAlarmXSet(DiagInterface.AlarmCore,'EventIDCode.12297');
		12298:  AlarmCount[71] := AlarmCount[71] + 1; MpAlarmXSet(DiagInterface.AlarmCore,'EventIDCode.12298');
		12299:  AlarmCount[72] := AlarmCount[72] + 1; MpAlarmXSet(DiagInterface.AlarmCore,'EventIDCode.12299');
		12300:  AlarmCount[73] := AlarmCount[73] + 1; MpAlarmXSet(DiagInterface.AlarmCore,'EventIDCode.12300');
		12301:  AlarmCount[74] := AlarmCount[74] + 1; MpAlarmXSet(DiagInterface.AlarmCore,'EventIDCode.12301');
		12302:  AlarmCount[75] := AlarmCount[75] + 1; MpAlarmXSet(DiagInterface.AlarmCore,'EventIDCode.12302');
		12303:  AlarmCount[76] := AlarmCount[76] + 1; MpAlarmXSet(DiagInterface.AlarmCore,'EventIDCode.12303');
		12304:  AlarmCount[77] := AlarmCount[77] + 1; MpAlarmXSet(DiagInterface.AlarmCore,'EventIDCode.12304');
		12305:  AlarmCount[78] := AlarmCount[78] + 1; MpAlarmXSet(DiagInterface.AlarmCore,'EventIDCode.12305');
		12307:  AlarmCount[79] := AlarmCount[79] + 1; MpAlarmXSet(DiagInterface.AlarmCore,'EventIDCode.12307');
		12312:  AlarmCount[80] := AlarmCount[80] + 1; MpAlarmXSet(DiagInterface.AlarmCore,'EventIDCode.12312');
		12313:  AlarmCount[81] := AlarmCount[81] + 1; MpAlarmXSet(DiagInterface.AlarmCore,'EventIDCode.12313');
		12314:  AlarmCount[82] := AlarmCount[82] + 1; MpAlarmXSet(DiagInterface.AlarmCore,'EventIDCode.12314');
		12315:  AlarmCount[83] := AlarmCount[83] + 1; MpAlarmXSet(DiagInterface.AlarmCore,'EventIDCode.12315');
		12316:  AlarmCount[84] := AlarmCount[84] + 1; MpAlarmXSet(DiagInterface.AlarmCore,'EventIDCode.12316');
		12317:  AlarmCount[85] := AlarmCount[85] + 1; MpAlarmXSet(DiagInterface.AlarmCore,'EventIDCode.12317');
		12320:  AlarmCount[86] := AlarmCount[86] + 1; MpAlarmXSet(DiagInterface.AlarmCore,'EventIDCode.12320');
		12322:  AlarmCount[87] := AlarmCount[87] + 1; MpAlarmXSet(DiagInterface.AlarmCore,'EventIDCode.12322');
		12323:  AlarmCount[88] := AlarmCount[88] + 1; MpAlarmXSet(DiagInterface.AlarmCore,'EventIDCode.12323');
		12328:  AlarmCount[89] := AlarmCount[89] + 1; MpAlarmXSet(DiagInterface.AlarmCore,'EventIDCode.12328');
		12330:  AlarmCount[90] := AlarmCount[90] + 1; MpAlarmXSet(DiagInterface.AlarmCore,'EventIDCode.12330');
		12331:  AlarmCount[91] := AlarmCount[91] + 1; MpAlarmXSet(DiagInterface.AlarmCore,'EventIDCode.12331');
		12333:  AlarmCount[92] := AlarmCount[92] + 1; MpAlarmXSet(DiagInterface.AlarmCore,'EventIDCode.12333');
		12334:  AlarmCount[93] := AlarmCount[93] + 1; MpAlarmXSet(DiagInterface.AlarmCore,'EventIDCode.12334');
		12335:  AlarmCount[94] := AlarmCount[94] + 1; MpAlarmXSet(DiagInterface.AlarmCore,'EventIDCode.12335');
		12336:  AlarmCount[95] := AlarmCount[95] + 1; MpAlarmXSet(DiagInterface.AlarmCore,'EventIDCode.12336');
		12337:  AlarmCount[96] := AlarmCount[96] + 1; MpAlarmXSet(DiagInterface.AlarmCore,'EventIDCode.12337');
		12338:  AlarmCount[97] := AlarmCount[97] + 1; MpAlarmXSet(DiagInterface.AlarmCore,'EventIDCode.12338');
		12340:  AlarmCount[98] := AlarmCount[98] + 1; MpAlarmXSet(DiagInterface.AlarmCore,'EventIDCode.12340');
		12341:  AlarmCount[99] := AlarmCount[99] + 1; MpAlarmXSet(DiagInterface.AlarmCore,'EventIDCode.12341');
		12342:  AlarmCount[100] := AlarmCount[100] + 1; MpAlarmXSet(DiagInterface.AlarmCore,'EventIDCode.12342');
		12343:  AlarmCount[101] := AlarmCount[101] + 1; MpAlarmXSet(DiagInterface.AlarmCore,'EventIDCode.12343');
		12344:  AlarmCount[102] := AlarmCount[102] + 1; MpAlarmXSet(DiagInterface.AlarmCore,'EventIDCode.12344');
		12345:  AlarmCount[103] := AlarmCount[103] + 1; MpAlarmXSet(DiagInterface.AlarmCore,'EventIDCode.12345');
		12346:  AlarmCount[104] := AlarmCount[104] + 1; MpAlarmXSet(DiagInterface.AlarmCore,'EventIDCode.12346');
		12347:  AlarmCount[105] := AlarmCount[105] + 1; MpAlarmXSet(DiagInterface.AlarmCore,'EventIDCode.12347');
		12348:  AlarmCount[106] := AlarmCount[106] + 1; MpAlarmXSet(DiagInterface.AlarmCore,'EventIDCode.12348');
		4007:   AlarmCount[107] := AlarmCount[107] + 1; MpAlarmXSet(DiagInterface.AlarmCore,'EventIDCode.4007');
		7230:   AlarmCount[108] := AlarmCount[108] + 1; MpAlarmXSet(DiagInterface.AlarmCore,'EventIDCode.7230');
		4005:   AlarmCount[109] := AlarmCount[109] + 1; MpAlarmXSet(DiagInterface.AlarmCore,'EventIDCode.4005');
		4098:   AlarmCount[110] := AlarmCount[110] + 1; MpAlarmXSet(DiagInterface.AlarmCore,'EventIDCode.4098');
		9106:   AlarmCount[111] := AlarmCount[111] + 1; MpAlarmXSet(DiagInterface.AlarmCore,'EventIDCode.9106');

		ELSE
			MpAlarmXSet(DiagInterface.AlarmCore,'EventIDCode.xxxx');
		END_CASE

END_ACTION
```

### Package Logical/Source/SampleTrak/Assembly - EquipmentModule1

### Assembly.var
```iecst
(*Shuttle initialization variables*)
VAR
	ShInit : SubroutineSequenceType;
	ShInitState : USINT;
	ShuttleUserData : ShuttleUserDataType;
	TrackInterface : ModuleInterfaceType;
	ModuleName : STRING[40];
END_VAR
```

### Assembly.typ
```iecst
TYPE
	TrakInterfaceType : 	STRUCT
		SampleTrak : McAssemblyType;
		ModulePml : MpComIdentType;
	END_STRUCT;
END_TYPE
```

### Program Logical/Source/SampleTrak/Assembly/AsmConfig (IEC)

#### Main.st
```iecst
PROGRAM _INIT
	(* Insert code here *)
	ModuleName := 'TrakModule';

	gRecipeXml_TrackModule;
	gTrakModule;

END_PROGRAM

PROGRAM _CYCLIC
	(* Insert code here *)

END_PROGRAM

PROGRAM _EXIT
	(* Insert code here *)

END_PROGRAM
```

### Program Logical/Source/SampleTrak/Assembly/AsmAlarm (IEC)

#### Variables.var
```iecst
VAR
	fbAlarmTrackModule : MpAlarmXCore;
	FilterConfiguration : STRING[1000] := '';
	SortConfiguration : STRING[1000] := '';
	HistoryFilter : STRING[2000] := '';
	HistorySort : STRING[2000] := '';
	TriggerTestAlarm : BOOL;
	TriggerTestWarning : BOOL;
	TriggerTestInformation : BOOL;
END_VAR
```

#### Main.st
```iecst
PROGRAM _INIT
	(* Insert code here *)
	FilterConfiguration;
	SortConfiguration;
	HistoryFilter;
	HistorySort;

END_PROGRAM

PROGRAM _CYCLIC
	(* Insert code here *)

	fbAlarmTrakModule(MpLink := ADR(gAlarmXCore_TrakModule), Enable := TRUE);

	TriggerTestAlarm;
	TriggerTestInformation;
	TriggerTestWarning;

	gAlarmXCore_EM2;
	gAlarmXCore_EM3;

END_PROGRAM

PROGRAM _EXIT
	(* Insert code here *)

END_PROGRAM
```

### Program Logical/Source/SampleTrak/Assembly/AsmSampleTrak (IEC)

#### Variables.var
```iecst
VAR
	AssemblyState : TrBaseAsmStateEnum;
	fbAsmReadStatus : MC_BR_AsmReadStatus_AcpTrak;
	fbAsmReadInfo : MC_BR_AsmReadInfo_AcpTrak;
	fbAsmPowerOn : MC_BR_AsmPowerOn_AcpTrak;
	fbAsmPowerOff : MC_BR_AsmPowerOff_AcpTrak;
	fbAsmReset : MC_BR_AsmReset_AcpTrak;
	fbTrakModule : MpPackMLModule;
	parTrakModule : MpPackMLModuleParType;
	TrakInterface : TrakInterfaceType;
END_VAR
```
